  MoveL 6540 to (-70.92, -30.3, -10) mm, rotated rx 180 ry 0 rz 90 deg; joints [72.111, -18.401, 88.578, 0, 19.823, 72.111]
  MoveC 6541 to (-72.65, -31.38, -10) mm, rotated rx 180 ry 0 rz 90 deg; joints [72.056, -18.422, 88.671, 0, 19.752, 72.056] to (-73.33, -33.3, -10) mm, rotated rx 180 ry 0 rz 90 deg; joints [71.985, -18.423, 88.674, 0, 19.749, 71.985]
  MoveL 6542 to (-73.33, -68.7, -10) mm, rotated rx 180 ry 0 rz 90 deg; joints [70.818, -18.238, 87.875, 0, 20.362, 70.818]
  MoveL 6543 to (-73.33, -69.73, -10) mm, rotated rx 180 ry 0 rz 90 deg; joints [70.785, -18.232, 87.851, 0, 20.381, 70.785]
  MoveC 6544 to (-72.43, -71.9, -10) mm, rotated rx -180 ry 0 rz 90 deg; joints [70.724, -18.206, 87.74, 0, 20.466, 70.724] to (-70.27, -72.81, -10) mm, rotated rx 180 ry 0 rz 90 deg; joints [70.719, -18.167, 87.574, 0, 20.593, 70.719]
  MoveL 6545 to (-69.65, -72.82, -10) mm, rotated rx 180 ry 0 rz 90 deg; joints [70.726, -18.157, 87.532, 0, 20.625, 70.726]
  MoveL 6546 to (-55.44, -72.67, -10) mm, rotated rx -180 ry 0 rz 90 deg; joints [70.891, -17.926, 86.573, 0, 21.353, 70.891]
  MoveL 6547 to (-54.49, -72.66, -10) mm, rotated rx -180 ry 0 rz 90 deg; joints [70.902, -17.91, 86.509, 0, 21.401, 70.902]
  MoveL 6548 to (-37.43, -72.45, -10) mm, rotated rx -180 ry 0 rz 90 deg; joints [71.098, -17.621, 85.344, 0, 22.277, 71.098]
  MoveL 6549 to (-36.13, -72.43, -10) mm, rotated rx 180 ry 0 rz 90 deg; joints [71.114, -17.599, 85.254, 0, 22.344, 71.114]
  MoveC 6550 to (-35.1, -72.24, -10) mm, rotated rx -180 ry 0 rz 90 deg; joints [71.131, -17.582, 85.188, 0, 22.394, 71.131] to (-34.2, -71.71, -10) mm, rotated rx -180 ry 0 rz 90 deg; joints [71.158, -17.569, 85.138, 0, 22.431, 71.158]
  MoveC 6551 to (-33.55, -70.97, -10) mm, rotated rx -180 ry 0 rz 90 deg; joints [71.188, -17.562, 85.111, 0, 22.452, 71.188] to (-33.16, -70.08, -10) mm, rotated rx 180 ry 0 rz 90 deg; joints [71.221, -17.561, 85.105, 0, 22.456, 71.221]
  MoveL 6552 to (-21.39, -24.64, -10) mm, rotated rx 180 ry 0 rz 90 deg; joints [72.81, -17.613, 85.312, 0, 22.301, 72.81]
  MoveL 6553 to (-21.34, -24.17, -10) mm, rotated rx 180 ry 0 rz 90 deg; joints [72.826, -17.615, 85.319, 0, 22.296, 72.826]
  MoveC 6554 to (-22.27, -22.08, -10) mm, rotated rx -180 ry 0 rz 90 deg; joints [72.884, -17.642, 85.428, 0, 22.214, 72.884] to (-24.17, -20.81, -10) mm, rotated rx 180 ry 0 rz 90 deg; joints [72.906, -17.682, 85.587, 0, 22.095, 72.906]
  MoveC 6555 to (-24.63, -20.72, -10) mm, rotated rx -180 ry 0 rz 90 deg; joints [72.905, -17.691, 85.622, 0, 22.069, 72.905] to (-25.11, -20.75, -10) mm, rotated rx 180 ry 0 rz 90 deg; joints [72.899, -17.699, 85.655, 0, 22.045, 72.899]
  MoveL 6556 to (-31.75, -22.12, -10) mm, rotated rx 180 ry 0 rz 90 deg; joints [72.788, -17.806, 86.085, 0, 21.721, 72.788]
  MoveL 6557 to (-48.02, -25.51, -10) mm, rotated rx 180 ry 0 rz 90 deg; joints [72.51, -18.061, 87.131, 0, 20.93, 72.51]
  MoveL 6558 to (-46.48, -32.9, -10) mm, rotated rx 180 ry 0 rz 90 deg; joints [72.284, -17.997, 86.865, 0, 21.132, 72.284]
  MoveL 6559 to (-46.48, -32.9, -7) mm, rotated rx 180 ry 0 rz 90 deg; joints [72.284, -18.152, 86.967, 0, 21.185, 72.284]
  Establecer velocidad (1000.0 mm/s)
  MoveL 6560 to (-46.48, -32.9, 10) mm, rotated rx 180 ry 0 rz 90 deg; joints [72.284, -19.031, 87.535, 0, 21.495, 72.284]
  Establecer velocidad (66.7 mm/s)
  MoveL 6561 to (15.27, -63.53, 10) mm, rotated rx 180 ry 0 rz 90 deg; joints [71.941, -17.71, 82.508, 0, 25.202, 71.941]
  MoveL 6562 to (15.27, -63.53, -6.75) mm, rotated rx 180 ry 0 rz 90 deg; joints [71.941, -16.862, 81.946, 0, 24.916, 71.941]
  MoveL 6563 to (15.14, -65.04, -7.16) mm, rotated rx -180 ry 0 rz 90 deg; joints [71.892, -16.834, 81.906, 0, 24.928, 71.892]
  MoveL 6564 to (15.37, -66.54, -7.56) mm, rotated rx -180 ry 0 rz 90 deg; joints [71.847, -16.8, 81.84, 0, 24.959, 71.847]
  MoveL 6565 to (15.92, -67.95, -7.97) mm, rotated rx -180 ry 0 rz 90 deg; joints [71.809, -16.759, 81.753, 0, 25.006, 71.809]
  MoveL 6566 to (16.78, -69.21, -8.37) mm, rotated rx 180 ry 0 rz 90 deg; joints [71.778, -16.713, 81.647, 0, 25.066, 71.778]
  MoveL 6567 to (17.89, -70.24, -8.78) mm, rotated rx 180 ry 0 rz 90 deg; joints [71.758, -16.663, 81.528, 0, 25.135, 71.758]
  MoveL 6568 to (19.21, -71.01, -9.19) mm, rotated rx -180 ry 0 rz 90 deg; joints [71.747, -16.611, 81.401, 0, 25.21, 71.747]
  MoveL 6569 to (20.66, -71.46, -9.59) mm, rotated rx 180 ry 0 rz 90 deg; joints [71.748, -16.559, 81.271, 0, 25.287, 71.748]
  MoveL 6570 to (22.17, -71.55, -10) mm, rotated rx 180 ry 0 rz 90 deg; joints [71.761, -16.507, 81.145, 0, 25.362, 71.761]
  MoveC 6571 to (32.54, -71.19, -10) mm, rotated rx -180 ry 0 rz 90 deg; joints [71.878, -16.297, 80.397, 0, 25.9, 71.878] to (42.91, -70.78, -10) mm, rotated rx -180 ry 0 rz 90 deg; joints [71.995, -16.083, 79.643, 0, 26.44, 71.995]
  MoveC 6572 to (45.2, -67.86, -10) mm, rotated rx -180 ry 0 rz 90 deg; joints [72.108, -16.055, 79.544, 0, 26.51, 72.108] to (45.35, -64.16, -10) mm, rotated rx 180 ry 0 rz 90 deg; joints [72.224, -16.077, 79.621, 0, 26.455, 72.224]
  MoveC 6573 to (34.71, -51.22, -10) mm, rotated rx -180 ry 0 rz 90 deg; joints [72.521, -16.385, 80.708, 0, 25.677, 72.521] to (23.95, -38.38, -10) mm, rotated rx -180 ry 0 rz 90 deg; joints [72.819, -16.684, 81.785, 0, 24.899, 72.819]
  MoveL 6574 to (22.88, -37.43, -10) mm, rotated rx 180 ry 0 rz 90 deg; joints [72.838, -16.711, 81.884, 0, 24.827, 72.838]
  MoveL 6575 to (21.72, -36.48, -10) mm, rotated rx 180 ry 0 rz 90 deg; joints [72.857, -16.739, 81.989, 0, 24.75, 72.857]
  MoveL 6576 to (13.74, -29.98, -10) mm, rotated rx -180 ry 0 rz 90 deg; joints [72.986, -16.934, 82.708, 0, 24.226, 72.986]
  MoveL 6577 to (13.21, -29.55, -10) mm, rotated rx 180 ry 0 rz 90 deg; joints [72.994, -16.947, 82.756, 0, 24.191, 72.994]
  MoveC 6578 to (10.33, -29.1, -10) mm, rotated rx 180 ry 0 rz 90 deg; joints [72.98, -17.005, 82.972, 0, 24.033, 72.98] to (7.97, -30.8, -10) mm, rotated rx 180 ry 0 rz 90 deg; joints [72.903, -17.04, 83.104, 0, 23.936, 72.903]
  MoveL 6579 to (7.68, -31.75, -10) mm, rotated rx 180 ry 0 rz 90 deg; joints [72.87, -17.04, 83.104, 0, 23.936, 72.87]
  MoveL 6580 to (-2.03, -67.76, -10) mm, rotated rx -180 ry 0 rz 90 deg; joints [71.628, -17.006, 82.975, 0, 24.031, 71.628]
  MoveL 6581 to (-2.14, -68.23, -10) mm, rotated rx 180 ry 0 rz 90 deg; joints [71.612, -17.005, 82.971, 0, 24.034, 71.612]
  MoveC 6582 to (-1.24, -70.97, -10) mm, rotated rx 180 ry 0 rz 90 deg; joints [71.535, -16.97, 82.842, 0, 24.128, 71.535] to (1.42, -72.1, -10) mm, rotated rx 180 ry 0 rz 90 deg; joints [71.528, -16.912, 82.626, 0, 24.286, 71.528]
  MoveC 6583 to (11.8, -71.85, -10) mm, rotated rx 180 ry 0 rz 90 deg; joints [71.644, -16.712, 81.888, 0, 24.824, 71.644] to (22.17, -71.55, -10) mm, rotated rx 180 ry 0 rz 90 deg; joints [71.761, -16.507, 81.145, 0, 25.362, 71.761]
  MoveL 6584 to (21.93, -64.01, -10) mm, rotated rx 180 ry 0 rz 90 deg; joints [71.994, -16.561, 81.342, 0, 25.22, 71.994]
  MoveL 6585 to (21.93, -64.01, -7) mm, rotated rx -180 ry 0 rz 90 deg; joints [71.994, -16.713, 81.444, 0, 25.269, 71.994]
  Establecer velocidad (1000.0 mm/s)
  MoveL 6586 to (21.93, -64.01, 10) mm, rotated rx 180 ry 0 rz 90 deg; joints [71.994, -17.572, 82.015, 0, 25.557, 71.994]
  Establecer velocidad (66.7 mm/s)
  MoveL 6587 to (35, 18.65, 10) mm, rotated rx 180 ry 0 rz 90 deg; joints [74.731, -17.808, 82.861, 0, 24.947, 74.731]
  MoveL 6588 to (35, 18.65, -6.75) mm, rotated rx 180 ry 0 rz 90 deg; joints [74.731, -16.959, 82.299, 0, 24.66, 74.731]
  MoveL 6589 to (35.18, 20.15, -7.16) mm, rotated rx -180 ry 0 rz 90 deg; joints [74.781, -16.943, 82.302, 0, 24.641, 74.781]
  MoveL 6590 to (34.99, 21.66, -7.56) mm, rotated rx -180 ry 0 rz 90 deg; joints [74.827, -16.934, 82.332, 0, 24.602, 74.827]
  MoveL 6591 to (34.47, 23.09, -7.97) mm, rotated rx -180 ry 0 rz 90 deg; joints [74.869, -16.931, 82.384, 0, 24.547, 74.869]
  MoveL 6592 to (33.65, 24.37, -8.37) mm, rotated rx 180 ry 0 rz 90 deg; joints [74.902, -16.934, 82.455, 0, 24.479, 74.902]
  MoveL 6593 to (32.57, 25.43, -8.78) mm, rotated rx 180 ry 0 rz 90 deg; joints [74.927, -16.94, 82.541, 0, 24.399, 74.927]
  MoveL 6594 to (31.28, 26.23, -9.19) mm, rotated rx -180 ry 0 rz 90 deg; joints [74.941, -16.949, 82.637, 0, 24.312, 74.941]
  MoveL 6595 to (29.84, 26.72, -9.59) mm, rotated rx -180 ry 0 rz 90 deg; joints [74.945, -16.959, 82.737, 0, 24.222, 74.945]
  MoveL 6596 to (28.33, 26.86, -10) mm, rotated rx -180 ry 0 rz 90 deg; joints [74.936, -16.968, 82.835, 0, 24.133, 74.936]
  MoveC 6597 to (20.56, 26.8, -10) mm, rotated rx -180 ry 0 rz 90 deg; joints [74.867, -17.117, 83.395, 0, 23.723, 74.867] to (12.79, 26.71, -10) mm, rotated rx 180 ry 0 rz 90 deg; joints [74.796, -17.264, 83.95, 0, 23.313, 74.796]
  MoveC 6598 to (10.39, 25.38, -10) mm, rotated rx 180 ry 0 rz 90 deg; joints [74.731, -17.302, 84.096, 0, 23.205, 74.731] to (9.6, 22.74, -10) mm, rotated rx 180 ry 0 rz 90 deg; joints [74.639, -17.303, 84.101, 0, 23.202, 74.639]
  MoveL 6599 to (9.74, 22.27, -10) mm, rotated rx 180 ry 0 rz 90 deg; joints [74.625, -17.298, 84.082, 0, 23.216, 74.625]
  MoveL 6600 to (13.74, 11.38, -10) mm, rotated rx -180 ry 0 rz 90 deg; joints [74.309, -17.166, 83.579, 0, 23.587, 74.309]
  MoveL 6601 to (13.93, 10.89, -10) mm, rotated rx 180 ry 0 rz 90 deg; joints [74.295, -17.16, 83.556, 0, 23.604, 74.295]
  MoveC 6602 to (14.41, 10.01, -10) mm, rotated rx 180 ry 0 rz 90 deg; joints [74.271, -17.146, 83.504, 0, 23.643, 74.271] to (15.12, 9.3, -10) mm, rotated rx 180 ry 0 rz 90 deg; joints [74.255, -17.129, 83.438, 0, 23.691, 74.255]
  MoveL 6603 to (27.96, -0.34, -10) mm, rotated rx 180 ry 0 rz 90 deg; joints [74.063, -16.828, 82.315, 0, 24.513, 74.063]
  MoveL 6604 to (28.42, -0.67, -10) mm, rotated rx 180 ry 0 rz 90 deg; joints [74.056, -16.817, 82.274, 0, 24.543, 74.056]
  MoveC 6605 to (29.07, -1.02, -10) mm, rotated rx 180 ry 0 rz 90 deg; joints [74.051, -16.802, 82.22, 0, 24.583, 74.051] to (29.8, -1.18, -10) mm, rotated rx 180 ry 0 rz 90 deg; joints [74.053, -16.787, 82.164, 0, 24.623, 74.053]
  MoveC 6606 to (31.81, -0.82, -10) mm, rotated rx -180 ry 0 rz 90 deg; joints [74.082, -16.749, 82.025, 0, 24.724, 74.082] to (33.4, 0.47, -10) mm, rotated rx 180 ry 0 rz 90 deg; joints [74.138, -16.725, 81.936, 0, 24.789, 74.138]
  MoveL 6607 to (45.89, 18.48, -10) mm, rotated rx -180 ry 0 rz 90 deg; joints [74.82, -16.574, 81.388, 0, 25.187, 74.82]
  MoveL 6608 to (47.25, 20.51, -10) mm, rotated rx 180 ry 0 rz 90 deg; joints [74.896, -16.557, 81.327, 0, 25.23, 74.896]
  MoveC 6609 to (47.11, 23.56, -10) mm, rotated rx 180 ry 0 rz 90 deg; joints [74.992, -16.577, 81.398, 0, 25.179, 74.992] to (45.53, 26.17, -10) mm, rotated rx 180 ry 0 rz 90 deg; joints [75.062, -16.623, 81.566, 0, 25.057, 75.062]
  MoveC 6610 to (44.76, 26.68, -10) mm, rotated rx 180 ry 0 rz 90 deg; joints [75.071, -16.642, 81.633, 0, 25.009, 75.071] to (43.86, 26.86, -10) mm, rotated rx -180 ry 0 rz 90 deg; joints [75.069, -16.661, 81.702, 0, 24.959, 75.069]
  MoveC 6611 to (36.09, 26.87, -10) mm, rotated rx 180 ry 0 rz 90 deg; joints [75.004, -16.816, 82.271, 0, 24.545, 75.004] to (28.33, 26.86, -10) mm, rotated rx -180 ry 0 rz 90 deg; joints [74.936, -16.968, 82.835, 0, 24.133, 74.936]
  MoveL 6612 to (28.36, 19.31, -10) mm, rotated rx 180 ry 0 rz 90 deg; joints [74.694, -16.928, 82.684, 0, 24.244, 74.694]
  MoveL 6613 to (28.36, 19.31, -7) mm, rotated rx 180 ry 0 rz 90 deg; joints [74.694, -17.08, 82.786, 0, 24.294, 74.694]
  Establecer velocidad (1000.0 mm/s)
  MoveL 6614 to (28.36, 19.31, 10) mm, rotated rx 180 ry 0 rz 90 deg; joints [74.694, -17.944, 83.356, 0, 24.588, 74.694]
  Establecer velocidad (66.7 mm/s)
  MoveL 6615 to (6.83, 65.57, 10) mm, rotated rx 180 ry 0 rz 90 deg; joints [76.013, -18.584, 85.767, 0, 22.817, 76.013]
  MoveL 6616 to (6.83, 65.57, -6.75) mm, rotated rx -180 ry 0 rz 90 deg; joints [76.013, -17.726, 85.207, 0, 22.518, 76.013]
  MoveL 6617 to (6.78, 64.06, -7.16) mm, rotated rx 180 ry 0 rz 90 deg; joints [75.963, -17.699, 85.17, 0, 22.529, 75.963]
  MoveL 6618 to (7.11, 62.57, -7.56) mm, rotated rx 180 ry 0 rz 90 deg; joints [75.917, -17.665, 85.107, 0, 22.559, 75.917]
  MoveL 6619 to (7.75, 61.2, -7.97) mm, rotated rx -180 ry 0 rz 90 deg; joints [75.877, -17.626, 85.022, 0, 22.604, 75.877]
  MoveL 6620 to (8.69, 59.99, -8.37) mm, rotated rx -180 ry 0 rz 90 deg; joints [75.845, -17.583, 84.921, 0, 22.662, 75.845]
  MoveL 6621 to (9.86, 59.03, -8.78) mm, rotated rx 180 ry 0 rz 90 deg; joints [75.824, -17.537, 84.806, 0, 22.731, 75.824]
  MoveL 6622 to (11.22, 58.35, -9.19) mm, rotated rx 180 ry 0 rz 90 deg; joints [75.813, -17.488, 84.683, 0, 22.805, 75.813]
  MoveL 6623 to (12.7, 57.99, -9.59) mm, rotated rx -180 ry 0 rz 90 deg; joints [75.813, -17.438, 84.557, 0, 22.881, 75.813]
  MoveL 6624 to (14.21, 58, -10) mm, rotated rx 180 ry 0 rz 90 deg; joints [75.826, -17.389, 84.435, 0, 22.954, 75.826]
  MoveL 6625 to (16.31, 58.19, -10) mm, rotated rx 180 ry 0 rz 90 deg; joints [75.849, -17.352, 84.289, 0, 23.063, 75.849]
  MoveC 6626 to (25.93, 59.17, -10) mm, rotated rx -180 ry 0 rz 90 deg; joints [75.96, -17.176, 83.615, 0, 23.561, 75.96] to (35.54, 60.24, -10) mm, rotated rx -180 ry 0 rz 90 deg; joints [76.072, -16.996, 82.938, 0, 24.058, 76.072]
  MoveC 6627 to (46.2, 61.66, -10) mm, rotated rx -180 ry 0 rz 90 deg; joints [76.202, -16.793, 82.185, 0, 24.608, 76.202] to (56.82, 63.37, -10) mm, rotated rx 180 ry 0 rz 90 deg; joints [76.34, -16.586, 81.432, 0, 25.154, 76.34]
  MoveL 6628 to (56.82, 69.31, -10) mm, rotated rx 180 ry 0 rz 90 deg; joints [76.531, -16.616, 81.538, 0, 25.077, 76.531]
  MoveC 6629 to (39.09, 70.56, -10) mm, rotated rx 180 ry 0 rz 90 deg; joints [76.434, -16.976, 82.864, 0, 24.112, 76.434] to (21.32, 71.33, -10) mm, rotated rx -180 ry 0 rz 90 deg; joints [76.319, -17.319, 84.163, 0, 23.156, 76.319]
  MoveC 6630 to (0.83, 71.9, -10) mm, rotated rx -180 ry 0 rz 90 deg; joints [76.173, -17.694, 85.632, 0, 22.061, 76.173] to (-19.66, 72.35, -10) mm, rotated rx 180 ry 0 rz 90 deg; joints [76.019, -18.048, 87.076, 0, 20.972, 76.019]
  MoveC 6631 to (-22, 69.47, -10) mm, rotated rx -180 ry 0 rz 90 deg; joints [75.904, -18.075, 87.189, 0, 20.886, 75.904] to (-21.68, 65.78, -10) mm, rotated rx 180 ry 0 rz 90 deg; joints [75.783, -18.054, 87.103, 0, 20.952, 75.783]
  MoveL 6632 to (-7.47, 56.63, -10) mm, rotated rx 180 ry 0 rz 90 deg; joints [75.599, -17.772, 85.947, 0, 21.825, 75.599]
  MoveC 6633 to (-7.12, 56.43, -10) mm, rotated rx 180 ry 0 rz 90 deg; joints [75.596, -17.765, 85.919, 0, 21.846, 75.596] to (-6.75, 56.27, -10) mm, rotated rx -180 ry 0 rz 90 deg; joints [75.594, -17.758, 85.89, 0, 21.868, 75.594]
  MoveC 6634 to (4.78, 57.16, -10) mm, rotated rx 180 ry 0 rz 90 deg; joints [75.72, -17.557, 85.092, 0, 22.466, 75.72] to (16.31, 58.19, -10) mm, rotated rx 180 ry 0 rz 90 deg; joints [75.849, -17.352, 84.289, 0, 23.063, 75.849]
  MoveL 6635 to (15.59, 65.71, -10) mm, rotated rx 180 ry 0 rz 90 deg; joints [76.089, -17.4, 84.475, 0, 22.925, 76.089]
  MoveL 6636 to (0.19, 64.36, -10) mm, rotated rx 180 ry 0 rz 90 deg; joints [75.919, -17.672, 85.546, 0, 22.126, 75.919]
  MoveL 6637 to (0.19, 64.36, -7) mm, rotated rx 180 ry 0 rz 90 deg; joints [75.919, -17.826, 85.648, 0, 22.179, 75.919]
  Establecer velocidad (1000.0 mm/s)
  MoveL 6638 to (0.19, 64.36, 10) mm, rotated rx -180 ry 0 rz 90 deg; joints [75.919, -18.7, 86.216, 0, 22.484, 75.919]
  Establecer velocidad (66.7 mm/s)
  MoveL 6639 to (3.74, 65.44, 10) mm, rotated rx -180 ry 0 rz 90 deg; joints [75.983, -18.64, 85.984, 0, 22.656, 75.983]
  MoveL 6640 to (3.74, 65.44, -7) mm, rotated rx -180 ry 0 rz 90 deg; joints [75.983, -17.768, 85.415, 0, 22.352, 75.983]
  MoveL 6641 to (3.7, 63.92, -7.41) mm, rotated rx -180 ry 0 rz 90 deg; joints [75.933, -17.741, 85.378, 0, 22.363, 75.933]
  MoveL 6642 to (4.03, 62.44, -7.81) mm, rotated rx 180 ry 0 rz 90 deg; joints [75.887, -17.707, 85.314, 0, 22.393, 75.887]
  MoveL 6643 to (4.67, 61.06, -8.22) mm, rotated rx -180 ry 0 rz 90 deg; joints [75.847, -17.669, 85.23, 0, 22.438, 75.847]
  MoveL 6644 to (5.61, 59.86, -8.63) mm, rotated rx 180 ry 0 rz 90 deg; joints [75.816, -17.625, 85.129, 0, 22.497, 75.816]
  MoveL 6645 to (6.78, 58.9, -9.03) mm, rotated rx -180 ry 0 rz 90 deg; joints [75.794, -17.579, 85.014, 0, 22.565, 75.794]
  MoveL 6646 to (8.14, 58.22, -9.44) mm, rotated rx 180 ry 0 rz 90 deg; joints [75.783, -17.53, 84.891, 0, 22.639, 75.783]
  MoveL 6647 to (9.62, 57.86, -9.84) mm, rotated rx 180 ry 0 rz 90 deg; joints [75.783, -17.481, 84.766, 0, 22.715, 75.783]
  MoveL 6648 to (11.13, 57.87, -10.25) mm, rotated rx -180 ry 0 rz 90 deg; joints [75.796, -17.433, 84.644, 0, 22.788, 75.796]
  MoveL 6649 to (16.29, 58.36, -10.25) mm, rotated rx -180 ry 0 rz 90 deg; joints [75.855, -17.34, 84.285, 0, 23.055, 75.855]
  MoveC 6650 to (25.45, 59.31, -10.25) mm, rotated rx -180 ry 0 rz 90 deg; joints [75.96, -17.173, 83.644, 0, 23.529, 75.96] to (34.59, 60.34, -10.25) mm, rotated rx -180 ry 0 rz 90 deg; joints [76.068, -17.002, 83, 0, 24.002, 76.068]
  MoveC 6651 to (44.29, 61.63, -10.25) mm, rotated rx -180 ry 0 rz 90 deg; joints [76.187, -16.818, 82.315, 0, 24.502, 76.187] to (53.96, 63.16, -10.25) mm, rotated rx -180 ry 0 rz 90 deg; joints [76.312, -16.631, 81.631, 0, 25, 76.312]
  MoveL 6652 to (53.96, 69.23, -10.25) mm, rotated rx 180 ry 0 rz 90 deg; joints [76.506, -16.661, 81.74, 0, 24.921, 76.506]
  MoveC 6653 to (38.5, 70.34, -10.25) mm, rotated rx -180 ry 0 rz 90 deg; joints [76.422, -16.974, 82.894, 0, 24.08, 76.422] to (23.02, 71.05, -10.25) mm, rotated rx -180 ry 0 rz 90 deg; joints [76.323, -17.273, 84.027, 0, 23.246, 76.323]
  MoveC 6654 to (1.99, 71.66, -10.25) mm, rotated rx -180 ry 0 rz 90 deg; joints [76.174, -17.659, 85.538, 0, 22.121, 76.174] to (-19.04, 72.14, -10.25) mm, rotated rx 180 ry 0 rz 90 deg; joints [76.017, -18.024, 87.021, 0, 21.002, 76.017]
  MoveC 6655 to (-21.35, 69.3, -10.25) mm, rotated rx -180 ry 0 rz 90 deg; joints [75.903, -18.051, 87.132, 0, 20.918, 75.903] to (-21.05, 65.65, -10.25) mm, rotated rx 180 ry 0 rz 90 deg; joints [75.784, -18.03, 87.048, 0, 20.983, 75.784]
  MoveL 6656 to (-6.9, 56.54, -10.25) mm, rotated rx 180 ry 0 rz 90 deg; joints [75.601, -17.749, 85.897, 0, 21.852, 75.601]
  MoveC 6657 to (-6.66, 56.43, -10.25) mm, rotated rx 180 ry 0 rz 90 deg; joints [75.6, -17.744, 85.878, 0, 21.866, 75.6] to (-6.41, 56.41, -10.25) mm, rotated rx 180 ry 0 rz 90 deg; joints [75.601, -17.74, 85.86, 0, 21.88, 75.601]
  MoveC 6658 to (4.95, 57.32, -10.25) mm, rotated rx -180 ry 0 rz 90 deg; joints [75.726, -17.542, 85.074, 0, 22.468, 75.726] to (16.29, 58.36, -10.25) mm, rotated rx -180 ry 0 rz 90 deg; joints [75.855, -17.34, 84.285, 0, 23.055, 75.855]
  MoveL 6659 to (15.55, 65.87, -10.25) mm, rotated rx 180 ry 0 rz 90 deg; joints [76.094, -17.388, 84.472, 0, 22.916, 76.094]
  MoveL 6660 to (-3.03, 64.24, -10.25) mm, rotated rx 180 ry 0 rz 90 deg; joints [75.888, -17.715, 85.762, 0, 21.953, 75.888]
  MoveL 6661 to (-3.03, 64.24, -7.25) mm, rotated rx 180 ry 0 rz 90 deg; joints [75.888, -17.87, 85.864, 0, 22.006, 75.888]
  Establecer velocidad (1000.0 mm/s)
  MoveL 6662 to (-3.03, 64.24, 10) mm, rotated rx -180 ry 0 rz 90 deg; joints [75.888, -18.757, 86.441, 0, 22.316, 75.888]
  Establecer velocidad (66.7 mm/s)
  MoveL 6663 to (35.09, 18.39, 10) mm, rotated rx 180 ry 0 rz 90 deg; joints [74.724, -17.805, 82.849, 0, 24.956, 74.724]
  MoveL 6664 to (35.09, 18.39, -7) mm, rotated rx -180 ry 0 rz 90 deg; joints [74.724, -16.943, 82.279, 0, 24.664, 74.724]
  MoveL 6665 to (35.27, 19.9, -7.41) mm, rotated rx -180 ry 0 rz 90 deg; joints [74.773, -16.927, 82.282, 0, 24.645, 74.773]
  MoveL 6666 to (35.09, 21.41, -7.81) mm, rotated rx 180 ry 0 rz 90 deg; joints [74.82, -16.918, 82.312, 0, 24.607, 74.82]
  MoveL 6667 to (34.57, 22.84, -8.22) mm, rotated rx -180 ry 0 rz 90 deg; joints [74.861, -16.915, 82.363, 0, 24.552, 74.861]
  MoveL 6668 to (33.75, 24.12, -8.63) mm, rotated rx -180 ry 0 rz 90 deg; joints [74.895, -16.918, 82.435, 0, 24.483, 74.895]
  MoveL 6669 to (32.67, 25.19, -9.03) mm, rotated rx -180 ry 0 rz 90 deg; joints [74.92, -16.924, 82.52, 0, 24.404, 74.92]
  MoveL 6670 to (31.38, 25.99, -9.44) mm, rotated rx 180 ry 0 rz 90 deg; joints [74.935, -16.933, 82.616, 0, 24.317, 74.935]
  MoveL 6671 to (29.94, 26.48, -9.84) mm, rotated rx 180 ry 0 rz 90 deg; joints [74.938, -16.943, 82.716, 0, 24.227, 74.938]
  MoveL 6672 to (28.43, 26.62, -10.25) mm, rotated rx -180 ry 0 rz 90 deg; joints [74.929, -16.952, 82.815, 0, 24.138, 74.929]
  MoveC 6673 to (21.08, 26.58, -10.25) mm, rotated rx -180 ry 0 rz 90 deg; joints [74.864, -17.094, 83.344, 0, 23.749, 74.864] to (13.74, 26.52, -10.25) mm, rotated rx 180 ry 0 rz 90 deg; joints [74.798, -17.232, 83.87, 0, 23.362, 74.798]
  MoveL 6674 to (12.79, 26.47, -10.25) mm, rotated rx 180 ry 0 rz 90 deg; joints [74.788, -17.25, 83.937, 0, 23.312, 74.788]
  MoveC 6675 to (10.55, 25.01, -10.25) mm, rotated rx 180 ry 0 rz 90 deg; joints [74.721, -17.284, 84.069, 0, 23.215, 74.721] to (9.95, 22.4, -10.25) mm, rotated rx -180 ry 0 rz 90 deg; joints [74.631, -17.282, 84.061, 0, 23.221, 74.631]
  MoveL 6676 to (9.99, 22.27, -10.25) mm, rotated rx 180 ry 0 rz 90 deg; joints [74.627, -17.28, 84.055, 0, 23.225, 74.627]
  MoveL 6677 to (13.82, 11.85, -10.25) mm, rotated rx -180 ry 0 rz 90 deg; joints [74.325, -17.154, 83.574, 0, 23.58, 74.325]
  MoveL 6678 to (14.18, 10.92, -10.25) mm, rotated rx 180 ry 0 rz 90 deg; joints [74.298, -17.143, 83.53, 0, 23.612, 74.298]
  MoveC 6679 to (14.61, 10.13, -10.25) mm, rotated rx -180 ry 0 rz 90 deg; joints [74.277, -17.13, 83.483, 0, 23.647, 74.277] to (15.25, 9.5, -10.25) mm, rotated rx 180 ry 0 rz 90 deg; joints [74.262, -17.115, 83.425, 0, 23.69, 74.262]
  MoveL 6680 to (28.34, -0.31, -10.25) mm, rotated rx 180 ry 0 rz 90 deg; joints [74.067, -16.808, 82.279, 0, 24.529, 74.067]
  MoveC 6681 to (29.16, -0.73, -10.25) mm, rotated rx -180 ry 0 rz 90 deg; joints [74.061, -16.789, 82.211, 0, 24.579, 74.061] to (30.08, -0.84, -10.25) mm, rotated rx 180 ry 0 rz 90 deg; joints [74.066, -16.771, 82.142, 0, 24.629, 74.066]
  MoveL 6682 to (30.41, -0.82, -10.25) mm, rotated rx 180 ry 0 rz 90 deg; joints [74.07, -16.764, 82.118, 0, 24.646, 74.07]
  MoveC 6683 to (32.1, -0.33, -10.25) mm, rotated rx 180 ry 0 rz 90 deg; joints [74.101, -16.734, 82.006, 0, 24.728, 74.101] to (33.39, 0.86, -10.25) mm, rotated rx 180 ry 0 rz 90 deg; joints [74.15, -16.715, 81.936, 0, 24.779, 74.15]
  MoveL 6684 to (45.56, 18.48, -10.25) mm, rotated rx -180 ry 0 rz 90 deg; joints [74.817, -16.568, 81.403, 0, 25.165, 74.817]
  MoveL 6685 to (46.21, 19.43, -10.25) mm, rotated rx -180 ry 0 rz 90 deg; joints [74.853, -16.56, 81.374, 0, 25.186, 74.853]
  MoveL 6686 to (46.79, 20.37, -10.25) mm, rotated rx -180 ry 0 rz 90 deg; joints [74.888, -16.553, 81.35, 0, 25.203, 74.888]
  MoveC 6687 to (46.42, 23.91, -10.25) mm, rotated rx -180 ry 0 rz 90 deg; joints [74.997, -16.58, 81.448, 0, 25.133, 74.997] to (44.07, 26.58, -10.25) mm, rotated rx 180 ry 0 rz 90 deg; joints [75.062, -16.643, 81.673, 0, 24.97, 75.062]
  MoveC 6688 to (36.25, 26.62, -10.25) mm, rotated rx -180 ry 0 rz 90 deg; joints [74.997, -16.799, 82.246, 0, 24.553, 74.997] to (28.43, 26.62, -10.25) mm, rotated rx -180 ry 0 rz 90 deg; joints [74.929, -16.952, 82.815, 0, 24.138, 74.929]
  MoveL 6689 to (28.45, 19.07, -10.25) mm, rotated rx -180 ry 0 rz 90 deg; joints [74.687, -16.912, 82.664, 0, 24.248, 74.687]
  MoveL 6690 to (28.45, 19.07, -7.25) mm, rotated rx -180 ry 0 rz 90 deg; joints [74.687, -17.065, 82.767, 0, 24.298, 74.687]
  Establecer velocidad (1000.0 mm/s)
  MoveL 6691 to (28.45, 19.07, 10) mm, rotated rx -180 ry 0 rz 90 deg; joints [74.687, -17.941, 83.345, 0, 24.596, 74.687]
  Establecer velocidad (66.7 mm/s)
  MoveL 6692 to (15.14, -63.32, 10) mm, rotated rx -180 ry 0 rz 90 deg; joints [71.946, -17.714, 82.522, 0, 25.192, 71.946]
  MoveL 6693 to (15.14, -63.32, -7) mm, rotated rx -180 ry 0 rz 90 deg; joints [71.946, -16.853, 81.952, 0, 24.902, 71.946]
  MoveL 6694 to (15, -64.83, -7.41) mm, rotated rx -180 ry 0 rz 90 deg; joints [71.897, -16.826, 81.912, 0, 24.914, 71.897]
  MoveL 6695 to (15.23, -66.33, -7.81) mm, rotated rx -180 ry 0 rz 90 deg; joints [71.853, -16.791, 81.846, 0, 24.945, 71.853]
  MoveL 6696 to (15.8, -67.74, -8.22) mm, rotated rx 180 ry 0 rz 90 deg; joints [71.814, -16.75, 81.758, 0, 24.991, 71.814]
  MoveL 6697 to (16.65, -69, -8.63) mm, rotated rx 180 ry 0 rz 90 deg; joints [71.784, -16.704, 81.653, 0, 25.051, 71.784]
  MoveL 6698 to (17.77, -70.03, -9.03) mm, rotated rx -180 ry 0 rz 90 deg; joints [71.763, -16.654, 81.534, 0, 25.121, 71.763]
  MoveL 6699 to (19.08, -70.79, -9.44) mm, rotated rx 180 ry 0 rz 90 deg; joints [71.753, -16.602, 81.406, 0, 25.196, 71.753]
  MoveL 6700 to (20.53, -71.24, -9.84) mm, rotated rx 180 ry 0 rz 90 deg; joints [71.754, -16.55, 81.277, 0, 25.273, 71.754]
  MoveL 6701 to (22.05, -71.33, -10.25) mm, rotated rx -180 ry 0 rz 90 deg; joints [71.766, -16.498, 81.151, 0, 25.347, 71.766]
  MoveC 6702 to (32.24, -70.96, -10.25) mm, rotated rx 180 ry 0 rz 90 deg; joints [71.882, -16.293, 80.416, 0, 25.876, 71.882] to (42.43, -70.52, -10.25) mm, rotated rx 180 ry 0 rz 90 deg; joints [71.998, -16.082, 79.677, 0, 26.406, 71.998]
  MoveC 6703 to (44.68, -67.63, -10.25) mm, rotated rx 180 ry 0 rz 90 deg; joints [72.11, -16.055, 79.579, 0, 26.475, 72.11] to (44.82, -63.97, -10.25) mm, rotated rx 180 ry 0 rz 90 deg; joints [72.225, -16.077, 79.657, 0, 26.42, 72.225]
  MoveL 6704 to (44.11, -63.02, -10.25) mm, rotated rx -180 ry 0 rz 90 deg; joints [72.247, -16.098, 79.732, 0, 26.366, 72.247]
  MoveL 6705 to (37.89, -55.44, -10.25) mm, rotated rx 180 ry 0 rz 90 deg; joints [72.421, -16.279, 80.368, 0, 25.911, 72.421]
  MoveL 6706 to (24.12, -38.91, -10.25) mm, rotated rx 180 ry 0 rz 90 deg; joints [72.804, -16.664, 81.752, 0, 24.912, 72.804]
  MoveC 6707 to (23.68, -38.42, -10.25) mm, rotated rx -180 ry 0 rz 90 deg; joints [72.815, -16.676, 81.795, 0, 24.881, 72.815] to (23.2, -37.98, -10.25) mm, rotated rx 180 ry 0 rz 90 deg; joints [72.824, -16.688, 81.84, 0, 24.848, 72.824]
  MoveL 6708 to (22.54, -37.43, -10.25) mm, rotated rx -180 ry 0 rz 90 deg; joints [72.835, -16.705, 81.9, 0, 24.805, 72.835]
  MoveL 6709 to (13.27, -29.86, -10.25) mm, rotated rx -180 ry 0 rz 90 deg; joints [72.985, -16.932, 82.737, 0, 24.195, 72.985]
  MoveC 6710 to (11.38, -29.38, -10.25) mm, rotated rx 180 ry 0 rz 90 deg; joints [72.981, -16.971, 82.882, 0, 24.088, 72.981] to (9.49, -29.85, -10.25) mm, rotated rx -180 ry 0 rz 90 deg; joints [72.948, -17.004, 83.008, 0, 23.997, 72.948]
  MoveL 6711 to (9.16, -30.03, -10.25) mm, rotated rx 180 ry 0 rz 90 deg; joints [72.939, -17.009, 83.028, 0, 23.982, 72.939]
  MoveC 6712 to (8.42, -30.65, -10.25) mm, rotated rx 180 ry 0 rz 90 deg; joints [72.912, -17.02, 83.067, 0, 23.953, 72.912] to (7.99, -31.51, -10.25) mm, rotated rx 180 ry 0 rz 90 deg; joints [72.88, -17.023, 83.079, 0, 23.944, 72.88]
  MoveL 6713 to (-1.55, -66.81, -10.25) mm, rotated rx -180 ry 0 rz 90 deg; joints [71.663, -16.99, 82.954, 0, 24.036, 71.663]
  MoveL 6714 to (-1.89, -68.23, -10.25) mm, rotated rx -180 ry 0 rz 90 deg; joints [71.615, -16.987, 82.945, 0, 24.043, 71.615]
  MoveC 6715 to (-0.91, -70.83, -10.25) mm, rotated rx 180 ry 0 rz 90 deg; joints [71.543, -16.952, 82.813, 0, 24.139, 71.543] to (1.66, -71.88, -10.25) mm, rotated rx 180 ry 0 rz 90 deg; joints [71.537, -16.896, 82.605, 0, 24.291, 71.537]
  MoveC 6716 to (11.86, -71.64, -10.25) mm, rotated rx -180 ry 0 rz 90 deg; joints [71.651, -16.699, 81.88, 0, 24.819, 71.651] to (22.05, -71.33, -10.25) mm, rotated rx -180 ry 0 rz 90 deg; joints [71.766, -16.498, 81.151, 0, 25.347, 71.766]
  MoveL 6717 to (21.8, -63.78, -10.25) mm, rotated rx -180 ry 0 rz 90 deg; joints [72, -16.553, 81.348, 0, 25.205, 72]
  MoveL 6718 to (21.8, -63.78, -7.25) mm, rotated rx -180 ry 0 rz 90 deg; joints [72, -16.705, 81.451, 0, 25.254, 72]
  Establecer velocidad (1000.0 mm/s)
  MoveL 6719 to (21.8, -63.78, 10) mm, rotated rx 180 ry 0 rz 90 deg; joints [72, -17.577, 82.03, 0, 25.546, 72]
  Establecer velocidad (66.7 mm/s)
  MoveL 6720 to (-37.16, -52.05, 10) mm, rotated rx -180 ry 0 rz 90 deg; joints [71.759, -18.764, 86.468, 0, 22.296, 71.759]
  MoveL 6721 to (-37.16, -52.05, -7) mm, rotated rx 180 ry 0 rz 90 deg; joints [71.759, -17.89, 85.9, 0, 21.99, 71.759]
  MoveL 6722 to (-35.75, -52.61, -7.41) mm, rotated rx -180 ry 0 rz 90 deg; joints [71.756, -17.841, 85.776, 0, 22.065, 71.756]
  MoveL 6723 to (-34.24, -52.81, -7.81) mm, rotated rx 180 ry 0 rz 90 deg; joints [71.766, -17.793, 85.654, 0, 22.139, 71.766]
  MoveL 6724 to (-32.73, -52.67, -8.22) mm, rotated rx 180 ry 0 rz 90 deg; joints [71.786, -17.746, 85.538, 0, 22.208, 71.786]
  MoveL 6725 to (-31.28, -52.2, -8.63) mm, rotated rx -180 ry 0 rz 90 deg; joints [71.817, -17.703, 85.435, 0, 22.268, 71.817]
  MoveL 6726 to (-29.97, -51.43, -9.03) mm, rotated rx -180 ry 0 rz 90 deg; joints [71.855, -17.664, 85.348, 0, 22.315, 71.855]
  MoveL 6727 to (-28.87, -50.38, -9.44) mm, rotated rx 180 ry 0 rz 90 deg; joints [71.901, -17.63, 85.282, 0, 22.348, 71.901]
  MoveL 6728 to (-28.03, -49.12, -9.84) mm, rotated rx -180 ry 0 rz 90 deg; joints [71.95, -17.601, 85.238, 0, 22.363, 71.95]
  MoveL 6729 to (-27.52, -47.69, -10.25) mm, rotated rx 180 ry 0 rz 90 deg; joints [72.002, -17.579, 85.221, 0, 22.359, 72.002]
  MoveL 6730 to (-21.66, -25.11, -10.25) mm, rotated rx 180 ry 0 rz 90 deg; joints [72.792, -17.603, 85.312, 0, 22.29, 72.792]
  MoveC 6731 to (-21.58, -24.64, -10.25) mm, rotated rx 180 ry 0 rz 90 deg; joints [72.808, -17.604, 85.316, 0, 22.287, 72.808] to (-21.6, -24.17, -10.25) mm, rotated rx 180 ry 0 rz 90 deg; joints [72.823, -17.606, 85.328, 0, 22.279, 72.823]
  MoveC 6732 to (-22.64, -22.11, -10.25) mm, rotated rx 180 ry 0 rz 90 deg; joints [72.88, -17.636, 85.445, 0, 22.191, 72.88] to (-24.64, -20.94, -10.25) mm, rotated rx -180 ry 0 rz 90 deg; joints [72.897, -17.677, 85.609, 0, 22.068, 72.897]
  MoveC 6733 to (-25.03, -20.94, -10.25) mm, rotated rx 180 ry 0 rz 90 deg; joints [72.894, -17.684, 85.636, 0, 22.048, 72.894] to (-25.41, -20.99, -10.25) mm, rotated rx -180 ry 0 rz 90 deg; joints [72.888, -17.69, 85.662, 0, 22.029, 72.888]
  MoveL 6734 to (-32.69, -22.48, -10.25) mm, rotated rx -180 ry 0 rz 90 deg; joints [72.766, -17.808, 86.135, 0, 21.673, 72.766]
  MoveL 6735 to (-70.75, -30.41, -10.25) mm, rotated rx 180 ry 0 rz 90 deg; joints [72.109, -18.385, 88.555, 0, 19.829, 72.109]
  MoveC 6736 to (-72.48, -31.47, -10.25) mm, rotated rx -180 ry 0 rz 90 deg; joints [72.055, -18.406, 88.649, 0, 19.757, 72.055] to (-73.16, -33.39, -10.25) mm, rotated rx 180 ry 0 rz 90 deg; joints [71.984, -18.407, 88.653, 0, 19.754, 71.984]
  MoveL 6737 to (-73.17, -68.7, -10.25) mm, rotated rx -180 ry 0 rz 90 deg; joints [70.82, -18.222, 87.856, 0, 20.366, 70.82]
  MoveL 6738 to (-73.16, -69.64, -10.25) mm, rotated rx 180 ry 0 rz 90 deg; joints [70.79, -18.217, 87.833, 0, 20.384, 70.79]
  MoveC 6739 to (-72.23, -71.81, -10.25) mm, rotated rx 180 ry 0 rz 90 deg; joints [70.729, -18.19, 87.721, 0, 20.47, 70.729] to (-70.05, -72.68, -10.25) mm, rotated rx 180 ry 0 rz 90 deg; joints [70.726, -18.151, 87.553, 0, 20.598, 70.726]
  MoveL 6740 to (-38.38, -72.3, -10.25) mm, rotated rx 180 ry 0 rz 90 deg; joints [71.093, -17.626, 85.404, 0, 22.221, 71.093]
  MoveL 6741 to (-36.21, -72.27, -10.25) mm, rotated rx 180 ry 0 rz 90 deg; joints [71.118, -17.588, 85.256, 0, 22.333, 71.118]
  MoveC 6742 to (-34.5, -71.7, -10.25) mm, rotated rx -180 ry 0 rz 90 deg; joints [71.155, -17.562, 85.15, 0, 22.411, 71.155] to (-33.41, -70.25, -10.25) mm, rotated rx 180 ry 0 rz 90 deg; joints [71.213, -17.551, 85.109, 0, 22.442, 71.213]
  MoveC 6743 to (-33.25, -69.79, -10.25) mm, rotated rx -180 ry 0 rz 90 deg; joints [71.23, -17.551, 85.109, 0, 22.442, 71.23] to (-33.12, -69.31, -10.25) mm, rotated rx 180 ry 0 rz 90 deg; joints [71.246, -17.552, 85.111, 0, 22.441, 71.246]
  MoveL 6744 to (-27.52, -47.69, -10.25) mm, rotated rx 180 ry 0 rz 90 deg; joints [72.002, -17.579, 85.221, 0, 22.359, 72.002]
  MoveL 6745 to (-34.82, -45.8, -10.25) mm, rotated rx -180 ry 0 rz 90 deg; joints [71.986, -17.717, 85.77, 0, 21.947, 71.986]
  MoveL 6746 to (-34.82, -45.8, -7.25) mm, rotated rx 180 ry 0 rz 90 deg; joints [71.986, -17.872, 85.872, 0, 22, 71.986]
  Establecer velocidad (1000.0 mm/s)
  MoveL 6747 to (-34.82, -45.8, 10) mm, rotated rx -180 ry 0 rz 90 deg; joints [71.986, -18.759, 86.449, 0, 22.31, 71.986]
  Establecer velocidad (66.7 mm/s)
  MoveL 6748 to (-64.93, 36.02, 10) mm, rotated rx 180 ry 0 rz 90 deg; joints [74.395, -19.659, 90.186, 0, 19.473, 74.395]
  MoveL 6749 to (-64.93, 36.02, -7) mm, rotated rx 180 ry 0 rz 90 deg; joints [74.395, -18.77, 89.618, 0, 19.152, 74.395]
  MoveL 6750 to (-66.43, 36.2, -7.41) mm, rotated rx 180 ry 0 rz 90 deg; joints [74.387, -18.772, 89.709, 0, 19.063, 74.387]
  MoveL 6751 to (-67.94, 36.02, -7.81) mm, rotated rx -180 ry 0 rz 90 deg; joints [74.367, -18.772, 89.793, 0, 18.98, 74.367]
  MoveL 6752 to (-69.37, 35.51, -8.22) mm, rotated rx -180 ry 0 rz 90 deg; joints [74.336, -18.77, 89.865, 0, 18.905, 74.336]
  MoveL 6753 to (-70.66, 34.69, -8.63) mm, rotated rx 180 ry 0 rz 90 deg; joints [74.296, -18.764, 89.922, 0, 18.842, 74.296]
  MoveL 6754 to (-71.72, 33.61, -9.03) mm, rotated rx -180 ry 0 rz 90 deg; joints [74.249, -18.754, 89.959, 0, 18.795, 74.249]
  MoveL 6755 to (-72.53, 32.32, -9.44) mm, rotated rx 180 ry 0 rz 90 deg; joints [74.197, -18.739, 89.975, 0, 18.764, 74.197]
  MoveL 6756 to (-73.03, 30.89, -9.84) mm, rotated rx 180 ry 0 rz 90 deg; joints [74.144, -18.719, 89.967, 0, 18.752, 74.144]
  MoveL 6757 to (-73.17, 29.38, -10.25) mm, rotated rx -180 ry 0 rz 90 deg; joints [74.091, -18.694, 89.934, 0, 18.76, 74.091]
  MoveL 6758 to (-73.17, 3.32, -10.25) mm, rotated rx 180 ry 0 rz 90 deg; joints [73.211, -18.581, 89.423, 0, 19.158, 73.211]
  MoveL 6759 to (-73.16, 2.37, -10.25) mm, rotated rx 180 ry 0 rz 90 deg; joints [73.179, -18.577, 89.403, 0, 19.173, 73.179]
  MoveC 6760 to (-72.28, 0.17, -10.25) mm, rotated rx -180 ry 0 rz 90 deg; joints [73.114, -18.553, 89.3, 0, 19.254, 73.114] to (-70.13, -0.83, -10.25) mm, rotated rx 180 ry 0 rz 90 deg; joints [73.102, -18.516, 89.135, 0, 19.381, 73.102]
  MoveC 6761 to (-69.87, -0.82, -10.25) mm, rotated rx -180 ry 0 rz 90 deg; joints [73.105, -18.513, 89.118, 0, 19.395, 73.105] to (-69.61, -0.78, -10.25) mm, rotated rx 180 ry 0 rz 90 deg; joints [73.109, -18.509, 89.102, 0, 19.407, 73.109]
  MoveC 6762 to (-46.55, 4.59, -10.25) mm, rotated rx 180 ry 0 rz 90 deg; joints [73.519, -18.174, 87.65, 0, 20.524, 73.519] to (-23.51, 10.03, -10.25) mm, rotated rx -180 ry 0 rz 90 deg; joints [73.92, -17.817, 86.172, 0, 21.645, 73.92]
  MoveC 6763 to (-22.88, 10.2, -10.25) mm, rotated rx 180 ry 0 rz 90 deg; joints [73.932, -17.807, 86.132, 0, 21.675, 73.932] to (-22.27, 10.41, -10.25) mm, rotated rx 180 ry 0 rz 90 deg; joints [73.945, -17.798, 86.094, 0, 21.704, 73.945]
  MoveC 6764 to (-20.94, 11.84, -10.25) mm, rotated rx 180 ry 0 rz 90 deg; joints [74.004, -17.782, 86.03, 0, 21.752, 74.004] to (-20.54, 13.74, -10.25) mm, rotated rx -180 ry 0 rz 90 deg; joints [74.07, -17.784, 86.04, 0, 21.744, 74.07]
  MoveC 6765 to (-20.66, 14.22, -10.25) mm, rotated rx 180 ry 0 rz 90 deg; joints [74.085, -17.789, 86.057, 0, 21.731, 74.085] to (-20.81, 14.69, -10.25) mm, rotated rx -180 ry 0 rz 90 deg; joints [74.099, -17.794, 86.077, 0, 21.716, 74.099]
  MoveL 6766 to (-26.71, 31.25, -10.25) mm, rotated rx 180 ry 0 rz 90 deg; joints [74.59, -17.973, 86.809, 0, 21.163, 74.59]
  MoveC 6767 to (-27.09, 31.98, -10.25) mm, rotated rx 180 ry 0 rz 90 deg; joints [74.611, -17.982, 86.85, 0, 21.133, 74.611] to (-27.66, 32.59, -10.25) mm, rotated rx 180 ry 0 rz 90 deg; joints [74.626, -17.995, 86.9, 0, 21.094, 74.626]
  MoveC 6768 to (-27.96, 32.82, -10.25) mm, rotated rx -180 ry 0 rz 90 deg; joints [74.631, -18.001, 86.926, 0, 21.075, 74.631] to (-28.28, 33.04, -10.25) mm, rotated rx -180 ry 0 rz 90 deg; joints [74.635, -18.007, 86.952, 0, 21.055, 74.635]
  MoveL 6769 to (-33.64, 36.53, -10.25) mm, rotated rx 180 ry 0 rz 90 deg; joints [74.703, -18.112, 87.388, 0, 20.723, 74.703]
  MoveL 6770 to (-64.4, 56.39, -10.25) mm, rotated rx -180 ry 0 rz 90 deg; joints [75.092, -18.674, 89.845, 0, 18.829, 75.092]
  MoveL 6771 to (-68.7, 59.15, -10.25) mm, rotated rx 180 ry 0 rz 90 deg; joints [75.147, -18.748, 90.184, 0, 18.565, 75.147]
  MoveC 6772 to (-70.58, 59.22, -10.25) mm, rotated rx -180 ry 0 rz 90 deg; joints [75.132, -18.776, 90.31, 0, 18.465, 75.132] to (-72.21, 58.28, -10.25) mm, rotated rx 180 ry 0 rz 90 deg; joints [75.085, -18.796, 90.403, 0, 18.393, 75.085]
  MoveC 6773 to (-72.91, 57.44, -10.25) mm, rotated rx -180 ry 0 rz 90 deg; joints [75.05, -18.803, 90.434, 0, 18.368, 75.05] to (-73.16, 56.39, -10.25) mm, rotated rx 180 ry 0 rz 90 deg; joints [75.012, -18.802, 90.432, 0, 18.37, 75.012]
  MoveL 6774 to (-73.17, 55.91, -10.25) mm, rotated rx 180 ry 0 rz 90 deg; joints [74.996, -18.8, 90.424, 0, 18.376, 74.996]
  MoveL 6775 to (-73.17, 29.38, -10.25) mm, rotated rx -180 ry 0 rz 90 deg; joints [74.091, -18.694, 89.934, 0, 18.76, 74.091]
  MoveL 6776 to (-65.62, 29.38, -10.25) mm, rotated rx 180 ry 0 rz 90 deg; joints [74.164, -18.582, 89.428, 0, 19.154, 74.164]
  MoveL 6777 to (-65.62, 29.38, -7.25) mm, rotated rx -180 ry 0 rz 90 deg; joints [74.164, -18.739, 89.53, 0, 19.209, 74.164]
  Establecer velocidad (1000.0 mm/s)
  MoveL 6778 to (-65.62, 29.38, 10) mm, rotated rx 180 ry 0 rz 90 deg; joints [74.164, -19.641, 90.107, 0, 19.534, 74.164]
  Establecer velocidad (66.7 mm/s)
  MoveL 6779 to (-64.76, 36.02, 10) mm, rotated rx 180 ry 0 rz 90 deg; joints [74.397, -19.656, 90.175, 0, 19.481, 74.397]
  MoveL 6780 to (-64.76, 36.02, -7.25) mm, rotated rx 180 ry 0 rz 90 deg; joints [74.397, -18.754, 89.598, 0, 19.156, 74.397]
  MoveL 6781 to (-66.27, 36.2, -7.66) mm, rotated rx 180 ry 0 rz 90 deg; joints [74.389, -18.756, 89.689, 0, 19.067, 74.389]
  MoveL 6782 to (-67.78, 36.02, -8.06) mm, rotated rx 180 ry 0 rz 90 deg; joints [74.368, -18.757, 89.773, 0, 18.984, 74.368]
  MoveL 6783 to (-69.21, 35.51, -8.47) mm, rotated rx 180 ry 0 rz 90 deg; joints [74.337, -18.755, 89.846, 0, 18.909, 74.337]
  MoveL 6784 to (-70.49, 34.69, -8.87) mm, rotated rx -180 ry 0 rz 90 deg; joints [74.297, -18.749, 89.902, 0, 18.846, 74.297]
  MoveL 6785 to (-71.56, 33.61, -9.28) mm, rotated rx 180 ry 0 rz 90 deg; joints [74.25, -18.739, 89.94, 0, 18.799, 74.25]
  MoveL 6786 to (-72.36, 32.32, -9.69) mm, rotated rx 180 ry 0 rz 90 deg; joints [74.199, -18.724, 89.955, 0, 18.768, 74.199]
  MoveL 6787 to (-72.86, 30.89, -10.09) mm, rotated rx -180 ry 0 rz 90 deg; joints [74.145, -18.704, 89.948, 0, 18.756, 74.145]
  MoveL 6788 to (-73, 29.38, -10.5) mm, rotated rx 180 ry 0 rz 90 deg; joints [74.093, -18.678, 89.915, 0, 18.764, 74.093]
  MoveL 6789 to (-73, 3.32, -10.5) mm, rotated rx -180 ry 0 rz 90 deg; joints [73.212, -18.565, 89.403, 0, 19.162, 73.212]
  MoveL 6790 to (-72.99, 2.37, -10.5) mm, rotated rx -180 ry 0 rz 90 deg; joints [73.181, -18.561, 89.383, 0, 19.178, 73.181]
  MoveC 6791 to (-71.95, 0.17, -10.5) mm, rotated rx 180 ry 0 rz 90 deg; joints [73.117, -18.535, 89.269, 0, 19.266, 73.117] to (-69.65, -0.62, -10.5) mm, rotated rx -180 ry 0 rz 90 deg; joints [73.114, -18.497, 89.099, 0, 19.398, 73.114]
  MoveL 6792 to (-68.91, -0.47, -10.5) mm, rotated rx -180 ry 0 rz 90 deg; joints [73.127, -18.487, 89.052, 0, 19.434, 73.127]
  MoveC 6793 to (-46.06, 4.86, -10.5) mm, rotated rx -180 ry 0 rz 90 deg; joints [73.533, -18.154, 87.613, 0, 20.541, 73.533] to (-23.22, 10.27, -10.5) mm, rotated rx 180 ry 0 rz 90 deg; joints [73.931, -17.8, 86.148, 0, 21.652, 73.931]
  MoveC 6794 to (-22.12, 10.77, -10.5) mm, rotated rx 180 ry 0 rz 90 deg; joints [73.958, -17.784, 86.082, 0, 21.702, 73.958] to (-21.32, 11.66, -10.5) mm, rotated rx -180 ry 0 rz 90 deg; joints [73.995, -17.775, 86.044, 0, 21.73, 73.995]
  MoveC 6795 to (-20.77, 13.13, -10.5) mm, rotated rx 180 ry 0 rz 90 deg; joints [74.048, -17.772, 86.035, 0, 21.738, 74.048] to (-20.98, 14.69, -10.5) mm, rotated rx 180 ry 0 rz 90 deg; joints [74.097, -17.784, 86.08, 0, 21.703, 74.097]
  MoveL 6796 to (-26.82, 31.12, -10.5) mm, rotated rx 180 ry 0 rz 90 deg; joints [74.585, -17.961, 86.806, 0, 21.155, 74.585]
  MoveC 6797 to (-27.32, 32.02, -10.5) mm, rotated rx 180 ry 0 rz 90 deg; joints [74.61, -17.973, 86.858, 0, 21.116, 74.61] to (-28.08, 32.71, -10.5) mm, rotated rx 180 ry 0 rz 90 deg; joints [74.626, -17.989, 86.923, 0, 21.066, 74.626]
  MoveC 6798 to (-48.25, 45.8, -10.5) mm, rotated rx 180 ry 0 rz 90 deg; joints [74.88, -18.373, 88.552, 0, 19.821, 74.88] to (-68.46, 58.83, -10.5) mm, rotated rx -180 ry 0 rz 90 deg; joints [75.139, -18.73, 90.153, 0, 18.578, 75.139]
  MoveC 6799 to (-68.78, 58.99, -10.5) mm, rotated rx 180 ry 0 rz 90 deg; joints [75.141, -18.736, 90.177, 0, 18.559, 75.141] to (-69.13, 59.06, -10.5) mm, rotated rx -180 ry 0 rz 90 deg; joints [75.14, -18.741, 90.202, 0, 18.539, 75.14]
  MoveC 6800 to (-71.13, 58.68, -10.5) mm, rotated rx 180 ry 0 rz 90 deg; joints [75.109, -18.769, 90.329, 0, 18.439, 75.109] to (-72.66, 57.33, -10.5) mm, rotated rx 180 ry 0 rz 90 deg; joints [75.049, -18.785, 90.407, 0, 18.378, 75.049]
  MoveC 6801 to (-72.89, 56.88, -10.5) mm, rotated rx -180 ry 0 rz 90 deg; joints [75.031, -18.787, 90.415, 0, 18.372, 75.031] to (-72.99, 56.39, -10.5) mm, rotated rx -180 ry 0 rz 90 deg; joints [75.013, -18.786, 90.413, 0, 18.374, 75.013]
  MoveL 6802 to (-73, 55.91, -10.5) mm, rotated rx -180 ry 0 rz 90 deg; joints [74.997, -18.785, 90.405, 0, 18.38, 74.997]
  MoveL 6803 to (-73, 29.38, -10.5) mm, rotated rx 180 ry 0 rz 90 deg; joints [74.093, -18.678, 89.915, 0, 18.764, 74.093]
  MoveL 6804 to (-65.45, 29.38, -10.5) mm, rotated rx 180 ry 0 rz 90 deg; joints [74.165, -18.566, 89.409, 0, 19.158, 74.165]
  MoveL 6805 to (-65.45, 29.38, -7.5) mm, rotated rx -180 ry 0 rz 90 deg; joints [74.165, -18.723, 89.511, 0, 19.213, 74.165]
  Establecer velocidad (1000.0 mm/s)
  MoveL 6806 to (-65.45, 29.38, 10) mm, rotated rx 180 ry 0 rz 90 deg; joints [74.165, -19.638, 90.096, 0, 19.542, 74.165]
  Establecer velocidad (66.7 mm/s)
  MoveL 6807 to (-39.92, -32.58, 10) mm, rotated rx 180 ry 0 rz 90 deg; joints [72.363, -18.921, 87.093, 0, 21.828, 72.363]
  MoveL 6808 to (-39.92, -32.58, -7.25) mm, rotated rx -180 ry 0 rz 90 deg; joints [72.363, -18.031, 86.516, 0, 21.515, 72.363]
  MoveL 6809 to (-40.05, -31.07, -7.66) mm, rotated rx -180 ry 0 rz 90 deg; joints [72.411, -18.021, 86.544, 0, 21.477, 72.411]
  MoveL 6810 to (-40.53, -29.63, -8.06) mm, rotated rx -180 ry 0 rz 90 deg; joints [72.453, -18.015, 86.595, 0, 21.421, 72.453]
  MoveL 6811 to (-41.32, -28.33, -8.47) mm, rotated rx 180 ry 0 rz 90 deg; joints [72.487, -18.015, 86.664, 0, 21.351, 72.487]
  MoveL 6812 to (-42.38, -27.24, -8.87) mm, rotated rx -180 ry 0 rz 90 deg; joints [72.512, -18.017, 86.746, 0, 21.271, 72.512]
  MoveL 6813 to (-43.65, -26.41, -9.28) mm, rotated rx 180 ry 0 rz 90 deg; joints [72.526, -18.022, 86.837, 0, 21.184, 72.526]
  MoveL 6814 to (-45.08, -25.89, -9.69) mm, rotated rx 180 ry 0 rz 90 deg; joints [72.528, -18.027, 86.933, 0, 21.094, 72.528]
  MoveL 6815 to (-46.59, -25.69, -10.09) mm, rotated rx 180 ry 0 rz 90 deg; joints [72.519, -18.032, 87.026, 0, 21.006, 72.519]
  MoveL 6816 to (-48.09, -25.86, -10.5) mm, rotated rx -180 ry 0 rz 90 deg; joints [72.498, -18.035, 87.112, 0, 20.923, 72.498]
  MoveL 6817 to (-64.91, -29.34, -10.5) mm, rotated rx -180 ry 0 rz 90 deg; joints [72.207, -18.286, 88.177, 0, 20.109, 72.207]
  MoveL 6818 to (-70.6, -30.54, -10.5) mm, rotated rx 180 ry 0 rz 90 deg; joints [72.106, -18.369, 88.534, 0, 19.835, 72.106]
  MoveC 6819 to (-72.22, -31.46, -10.5) mm, rotated rx 180 ry 0 rz 90 deg; joints [72.058, -18.389, 88.623, 0, 19.766, 72.058] to (-72.97, -33.17, -10.5) mm, rotated rx 180 ry 0 rz 90 deg; joints [71.994, -18.392, 88.636, 0, 19.756, 71.994]
  MoveL 6820 to (-73, -33.64, -10.5) mm, rotated rx 180 ry 0 rz 90 deg; joints [71.978, -18.39, 88.627, 0, 19.763, 71.978]
  MoveL 6821 to (-73, -34.59, -10.5) mm, rotated rx 180 ry 0 rz 90 deg; joints [71.946, -18.385, 88.607, 0, 19.778, 71.946]
  MoveL 6822 to (-73, -68.7, -10.5) mm, rotated rx -180 ry 0 rz 90 deg; joints [70.822, -18.207, 87.836, 0, 20.37, 70.822]
  MoveL 6823 to (-72.99, -69.55, -10.5) mm, rotated rx 180 ry 0 rz 90 deg; joints [70.795, -18.202, 87.816, 0, 20.386, 70.795]
  MoveC 6824 to (-72.07, -71.67, -10.5) mm, rotated rx 180 ry 0 rz 90 deg; joints [70.736, -18.175, 87.704, 0, 20.472, 70.736] to (-69.91, -72.53, -10.5) mm, rotated rx 180 ry 0 rz 90 deg; joints [70.732, -18.136, 87.539, 0, 20.598, 70.732]
  MoveL 6825 to (-38.38, -72.14, -10.5) mm, rotated rx -180 ry 0 rz 90 deg; joints [71.098, -17.614, 85.4, 0, 22.214, 71.098]
  MoveL 6826 to (-36.33, -72.1, -10.5) mm, rotated rx -180 ry 0 rz 90 deg; joints [71.122, -17.578, 85.259, 0, 22.319, 71.122]
  MoveC 6827 to (-34.48, -71.44, -10.5) mm, rotated rx -180 ry 0 rz 90 deg; joints [71.163, -17.55, 85.147, 0, 22.403, 71.163] to (-33.4, -69.78, -10.5) mm, rotated rx 180 ry 0 rz 90 deg; joints [71.228, -17.541, 85.111, 0, 22.43, 71.228]
  MoveL 6828 to (-21.86, -25.25, -10.5) mm, rotated rx -180 ry 0 rz 90 deg; joints [72.786, -17.592, 85.314, 0, 22.278, 72.786]
  MoveC 6829 to (-21.8, -24.95, -10.5) mm, rotated rx -180 ry 0 rz 90 deg; joints [72.796, -17.593, 85.316, 0, 22.276, 72.796] to (-21.76, -24.64, -10.5) mm, rotated rx -180 ry 0 rz 90 deg; joints [72.806, -17.594, 85.321, 0, 22.273, 72.806]
  MoveC 6830 to (-22.57, -22.64, -10.5) mm, rotated rx 180 ry 0 rz 90 deg; joints [72.863, -17.619, 85.42, 0, 22.199, 72.863] to (-24.26, -21.32, -10.5) mm, rotated rx -180 ry 0 rz 90 deg; joints [72.889, -17.656, 85.566, 0, 22.09, 72.889]
  MoveC 6831 to (-24.91, -21.16, -10.5) mm, rotated rx -180 ry 0 rz 90 deg; joints [72.888, -17.668, 85.615, 0, 22.053, 72.888] to (-25.59, -21.2, -10.5) mm, rotated rx 180 ry 0 rz 90 deg; joints [72.879, -17.679, 85.661, 0, 22.019, 72.879]
  MoveL 6832 to (-29.85, -22.08, -10.5) mm, rotated rx 180 ry 0 rz 90 deg; joints [72.808, -17.748, 85.938, 0, 21.81, 72.808]
  MoveL 6833 to (-48.09, -25.86, -10.5) mm, rotated rx -180 ry 0 rz 90 deg; joints [72.498, -18.035, 87.112, 0, 20.923, 72.498]
  MoveL 6834 to (-46.56, -33.25, -10.5) mm, rotated rx 180 ry 0 rz 90 deg; joints [72.272, -17.971, 86.846, 0, 21.124, 72.272]
  MoveL 6835 to (-46.56, -33.25, -7.5) mm, rotated rx -180 ry 0 rz 90 deg; joints [72.272, -18.126, 86.948, 0, 21.178, 72.272]
  Establecer velocidad (1000.0 mm/s)
  MoveL 6836 to (-46.56, -33.25, 10) mm, rotated rx -180 ry 0 rz 90 deg; joints [72.272, -19.03, 87.534, 0, 21.497, 72.272]
  Establecer velocidad (66.7 mm/s)
  MoveL 6837 to (14.97, -63.1, 10) mm, rotated rx -180 ry 0 rz 90 deg; joints [71.951, -17.719, 82.54, 0, 25.179, 71.951]
  MoveL 6838 to (14.97, -63.1, -7.25) mm, rotated rx 180 ry 0 rz 90 deg; joints [71.951, -16.846, 81.961, 0, 24.885, 71.951]
  MoveL 6839 to (14.84, -64.61, -7.66) mm, rotated rx 180 ry 0 rz 90 deg; joints [71.903, -16.818, 81.921, 0, 24.897, 71.903]
  MoveL 6840 to (15.07, -66.11, -8.06) mm, rotated rx 180 ry 0 rz 90 deg; joints [71.858, -16.783, 81.855, 0, 24.928, 71.858]
  MoveL 6841 to (15.63, -67.52, -8.47) mm, rotated rx -180 ry 0 rz 90 deg; joints [71.819, -16.742, 81.767, 0, 24.975, 71.819]
  MoveL 6842 to (16.49, -68.77, -8.87) mm, rotated rx 180 ry 0 rz 90 deg; joints [71.789, -16.696, 81.661, 0, 25.035, 71.789]
  MoveL 6843 to (17.61, -69.81, -9.28) mm, rotated rx -180 ry 0 rz 90 deg; joints [71.768, -16.646, 81.542, 0, 25.104, 71.768]
  MoveL 6844 to (18.93, -70.57, -9.69) mm, rotated rx 180 ry 0 rz 90 deg; joints [71.758, -16.594, 81.415, 0, 25.18, 71.758]
  MoveL 6845 to (20.38, -71.02, -10.09) mm, rotated rx 180 ry 0 rz 90 deg; joints [71.759, -16.542, 81.285, 0, 25.257, 71.759]
  MoveL 6846 to (21.89, -71.1, -10.5) mm, rotated rx -180 ry 0 rz 90 deg; joints [71.772, -16.49, 81.159, 0, 25.331, 71.772]
  MoveC 6847 to (31.92, -70.72, -10.5) mm, rotated rx 180 ry 0 rz 90 deg; joints [71.886, -16.288, 80.437, 0, 25.851, 71.886] to (41.94, -70.27, -10.5) mm, rotated rx -180 ry 0 rz 90 deg; joints [72.001, -16.082, 79.71, 0, 26.372, 72.001]
  MoveC 6848 to (43.51, -68.8, -10.5) mm, rotated rx 180 ry 0 rz 90 deg; joints [72.062, -16.059, 79.63, 0, 26.429, 72.062] to (44.32, -66.81, -10.5) mm, rotated rx -180 ry 0 rz 90 deg; joints [72.132, -16.055, 79.617, 0, 26.438, 72.132]
  MoveC 6849 to (44.55, -65.08, -10.5) mm, rotated rx -180 ry 0 rz 90 deg; joints [72.188, -16.062, 79.641, 0, 26.421, 72.188] to (44.07, -63.41, -10.5) mm, rotated rx 180 ry 0 rz 90 deg; joints [72.235, -16.084, 79.717, 0, 26.367, 72.235]
  MoveC 6850 to (34.2, -51.34, -10.5) mm, rotated rx -180 ry 0 rz 90 deg; joints [72.512, -16.369, 80.726, 0, 25.643, 72.512] to (24.21, -39.38, -10.5) mm, rotated rx -180 ry 0 rz 90 deg; joints [72.79, -16.647, 81.726, 0, 24.92, 72.79]
  MoveC 6851 to (23.77, -38.87, -10.5) mm, rotated rx 180 ry 0 rz 90 deg; joints [72.802, -16.659, 81.77, 0, 24.889, 72.802] to (23.32, -38.38, -10.5) mm, rotated rx 180 ry 0 rz 90 deg; joints [72.813, -16.671, 81.814, 0, 24.857, 72.813]
  MoveL 6852 to (13.74, -30.52, -10.5) mm, rotated rx -180 ry 0 rz 90 deg; joints [72.968, -16.906, 82.68, 0, 24.226, 72.968]
  MoveL 6853 to (13.27, -30.16, -10.5) mm, rotated rx 180 ry 0 rz 90 deg; joints [72.975, -16.917, 82.721, 0, 24.196, 72.975]
  MoveC 6854 to (11.08, -29.76, -10.5) mm, rotated rx -180 ry 0 rz 90 deg; joints [72.967, -16.961, 82.887, 0, 24.074, 72.967] to (9, -30.56, -10.5) mm, rotated rx -180 ry 0 rz 90 deg; joints [72.921, -16.996, 83.018, 0, 23.978, 72.921]
  MoveC 6855 to (8.46, -31.12, -10.5) mm, rotated rx -180 ry 0 rz 90 deg; joints [72.897, -17.003, 83.045, 0, 23.959, 72.897] to (8.14, -31.84, -10.5) mm, rotated rx -180 ry 0 rz 90 deg; joints [72.872, -17.005, 83.052, 0, 23.953, 72.872]
  MoveL 6856 to (-1.52, -67.56, -10.5) mm, rotated rx 180 ry 0 rz 90 deg; joints [71.64, -16.972, 82.926, 0, 24.046, 71.64]
  MoveC 6857 to (-1.62, -68.25, -10.5) mm, rotated rx 180 ry 0 rz 90 deg; joints [71.617, -16.969, 82.917, 0, 24.053, 71.617] to (-1.56, -68.94, -10.5) mm, rotated rx 180 ry 0 rz 90 deg; joints [71.596, -16.964, 82.896, 0, 24.068, 71.596]
  MoveC 6858 to (-0.36, -70.91, -10.5) mm, rotated rx -180 ry 0 rz 90 deg; joints [71.546, -16.928, 82.764, 0, 24.165, 71.546] to (1.83, -71.66, -10.5) mm, rotated rx -180 ry 0 rz 90 deg; joints [71.546, -16.882, 82.59, 0, 24.292, 71.546]
  MoveC 6859 to (11.86, -71.41, -10.5) mm, rotated rx -180 ry 0 rz 90 deg; joints [71.658, -16.688, 81.877, 0, 24.811, 71.658] to (21.89, -71.1, -10.5) mm, rotated rx -180 ry 0 rz 90 deg; joints [71.772, -16.49, 81.159, 0, 25.331, 71.772]
  MoveL 6860 to (21.63, -63.56, -10.5) mm, rotated rx -180 ry 0 rz 90 deg; joints [72.005, -16.545, 81.357, 0, 25.188, 72.005]
  MoveL 6861 to (21.63, -63.56, -7.5) mm, rotated rx -180 ry 0 rz 90 deg; joints [72.005, -16.697, 81.46, 0, 25.237, 72.005]
  Establecer velocidad (1000.0 mm/s)
  MoveL 6862 to (21.63, -63.56, 10) mm, rotated rx 180 ry 0 rz 90 deg; joints [72.005, -17.582, 82.048, 0, 25.534, 72.005]
  Establecer velocidad (66.7 mm/s)
  MoveL 6863 to (35.03, 18.14, 10) mm, rotated rx 180 ry 0 rz 90 deg; joints [74.715, -17.805, 82.849, 0, 24.956, 74.715]
  MoveL 6864 to (35.03, 18.14, -7.25) mm, rotated rx -180 ry 0 rz 90 deg; joints [74.715, -16.93, 82.27, 0, 24.66, 74.715]
  MoveL 6865 to (35.21, 19.65, -7.66) mm, rotated rx -180 ry 0 rz 90 deg; joints [74.765, -16.914, 82.273, 0, 24.641, 74.765]
  MoveL 6866 to (35.03, 21.16, -8.06) mm, rotated rx -180 ry 0 rz 90 deg; joints [74.811, -16.905, 82.302, 0, 24.603, 74.811]
  MoveL 6867 to (34.51, 22.59, -8.47) mm, rotated rx -180 ry 0 rz 90 deg; joints [74.853, -16.902, 82.354, 0, 24.548, 74.853]
  MoveL 6868 to (33.7, 23.87, -8.87) mm, rotated rx 180 ry 0 rz 90 deg; joints [74.887, -16.905, 82.425, 0, 24.48, 74.887]
  MoveL 6869 to (32.62, 24.94, -9.28) mm, rotated rx 180 ry 0 rz 90 deg; joints [74.912, -16.911, 82.511, 0, 24.4, 74.912]
  MoveL 6870 to (31.33, 25.74, -9.69) mm, rotated rx 180 ry 0 rz 90 deg; joints [74.926, -16.92, 82.606, 0, 24.314, 74.926]
  MoveL 6871 to (29.89, 26.24, -10.09) mm, rotated rx 180 ry 0 rz 90 deg; joints [74.93, -16.93, 82.706, 0, 24.224, 74.93]
  MoveL 6872 to (28.38, 26.38, -10.5) mm, rotated rx -180 ry 0 rz 90 deg; joints [74.921, -16.939, 82.805, 0, 24.135, 74.921]
  MoveC 6873 to (21.06, 26.35, -10.5) mm, rotated rx 180 ry 0 rz 90 deg; joints [74.857, -17.08, 83.333, 0, 23.747, 74.857] to (13.74, 26.29, -10.5) mm, rotated rx -180 ry 0 rz 90 deg; joints [74.791, -17.218, 83.857, 0, 23.361, 74.791]
  MoveC 6874 to (11.07, 25.08, -10.5) mm, rotated rx 180 ry 0 rz 90 deg; joints [74.728, -17.262, 84.025, 0, 23.237, 74.728] to (10.25, 22.27, -10.5) mm, rotated rx 180 ry 0 rz 90 deg; joints [74.63, -17.263, 84.028, 0, 23.234, 74.63]
  MoveL 6875 to (10.44, 21.73, -10.5) mm, rotated rx -180 ry 0 rz 90 deg; joints [74.614, -17.256, 84.004, 0, 23.252, 74.614]
  MoveL 6876 to (14.08, 11.85, -10.5) mm, rotated rx -180 ry 0 rz 90 deg; joints [74.327, -17.137, 83.548, 0, 23.589, 74.327]
  MoveL 6877 to (14.4, 11, -10.5) mm, rotated rx -180 ry 0 rz 90 deg; joints [74.303, -17.126, 83.507, 0, 23.619, 74.303]
  MoveC 6878 to (14.81, 10.27, -10.5) mm, rotated rx 180 ry 0 rz 90 deg; joints [74.283, -17.115, 83.464, 0, 23.651, 74.283] to (15.39, 9.69, -10.5) mm, rotated rx -180 ry 0 rz 90 deg; joints [74.269, -17.1, 83.41, 0, 23.691, 74.269]
  MoveL 6879 to (16.29, 9, -10.5) mm, rotated rx 180 ry 0 rz 90 deg; joints [74.256, -17.08, 83.331, 0, 23.748, 74.256]
  MoveL 6880 to (28.33, 0.01, -10.5) mm, rotated rx -180 ry 0 rz 90 deg; joints [74.077, -16.797, 82.278, 0, 24.52, 74.077]
  MoveC 6881 to (28.91, -0.32, -10.5) mm, rotated rx 180 ry 0 rz 90 deg; joints [74.072, -16.784, 82.229, 0, 24.555, 74.072] to (29.55, -0.49, -10.5) mm, rotated rx -180 ry 0 rz 90 deg; joints [74.072, -16.77, 82.179, 0, 24.591, 74.072]
  MoveC 6882 to (31.68, -0.19, -10.5) mm, rotated rx 180 ry 0 rz 90 deg; joints [74.101, -16.73, 82.03, 0, 24.7, 74.101] to (33.33, 1.18, -10.5) mm, rotated rx -180 ry 0 rz 90 deg; joints [74.16, -16.705, 81.938, 0, 24.767, 74.16]
  MoveL 6883 to (45.24, 18.48, -10.5) mm, rotated rx 180 ry 0 rz 90 deg; joints [74.814, -16.562, 81.418, 0, 25.144, 74.814]
  MoveL 6884 to (46.28, 20.04, -10.5) mm, rotated rx -180 ry 0 rz 90 deg; joints [74.873, -16.549, 81.373, 0, 25.177, 74.873]
  MoveC 6885 to (46.04, 23.37, -10.5) mm, rotated rx -180 ry 0 rz 90 deg; joints [74.977, -16.572, 81.456, 0, 25.116, 74.977] to (44.07, 26.06, -10.5) mm, rotated rx 180 ry 0 rz 90 deg; joints [75.046, -16.627, 81.654, 0, 24.973, 75.046]
  MoveC 6886 to (43.56, 26.25, -10.5) mm, rotated rx 180 ry 0 rz 90 deg; joints [75.047, -16.638, 81.695, 0, 24.943, 75.047] to (43.02, 26.32, -10.5) mm, rotated rx 180 ry 0 rz 90 deg; joints [75.045, -16.649, 81.736, 0, 24.913, 75.045]
  MoveC 6887 to (35.7, 26.36, -10.5) mm, rotated rx -180 ry 0 rz 90 deg; joints [74.984, -16.796, 82.272, 0, 24.523, 74.984] to (28.38, 26.38, -10.5) mm, rotated rx -180 ry 0 rz 90 deg; joints [74.921, -16.939, 82.805, 0, 24.135, 74.921]
  MoveL 6888 to (28.39, 18.83, -10.5) mm, rotated rx 180 ry 0 rz 90 deg; joints [74.679, -16.899, 82.656, 0, 24.244, 74.679]
  MoveL 6889 to (28.39, 18.83, -7.5) mm, rotated rx 180 ry 0 rz 90 deg; joints [74.679, -17.052, 82.758, 0, 24.294, 74.679]
  Establecer velocidad (1000.0 mm/s)
  MoveL 6890 to (28.39, 18.83, 10) mm, rotated rx 180 ry 0 rz 90 deg; joints [74.679, -17.941, 83.345, 0, 24.596, 74.679]
  Establecer velocidad (66.7 mm/s)
  MoveL 6891 to (4.27, 58.51, 10) mm, rotated rx 180 ry 0 rz 90 deg; joints [75.76, -18.599, 85.823, 0, 22.776, 75.76]
  MoveL 6892 to (4.27, 58.51, -7.25) mm, rotated rx 180 ry 0 rz 90 deg; joints [75.76, -17.714, 85.246, 0, 22.468, 75.76]
  MoveL 6893 to (5.67, 57.92, -7.66) mm, rotated rx 180 ry 0 rz 90 deg; joints [75.752, -17.665, 85.122, 0, 22.543, 75.752]
  MoveL 6894 to (7.17, 57.69, -8.06) mm, rotated rx -180 ry 0 rz 90 deg; joints [75.757, -17.616, 84.998, 0, 22.619, 75.757]
  MoveL 6895 to (8.69, 57.79, -8.47) mm, rotated rx -180 ry 0 rz 90 deg; joints [75.773, -17.568, 84.878, 0, 22.69, 75.773]
  MoveL 6896 to (10.14, 58.23, -8.87) mm, rotated rx -180 ry 0 rz 90 deg; joints [75.8, -17.523, 84.768, 0, 22.755, 75.8]
  MoveL 6897 to (11.47, 58.98, -9.28) mm, rotated rx 180 ry 0 rz 90 deg; joints [75.835, -17.481, 84.674, 0, 22.808, 75.835]
  MoveL 6898 to (12.59, 60, -9.69) mm, rotated rx 180 ry 0 rz 90 deg; joints [75.878, -17.445, 84.598, 0, 22.846, 75.878]
  MoveL 6899 to (13.46, 61.25, -10.09) mm, rotated rx -180 ry 0 rz 90 deg; joints [75.926, -17.414, 84.544, 0, 22.869, 75.926]
  MoveL 6900 to (14, 62.66, -10.5) mm, rotated rx -180 ry 0 rz 90 deg; joints [75.976, -17.389, 84.517, 0, 22.872, 75.976]
  MoveL 6901 to (16.36, 71.03, -10.5) mm, rotated rx -180 ry 0 rz 90 deg; joints [76.269, -17.384, 84.496, 0, 22.888, 76.269]
  MoveC 6902 to (-1.03, 71.54, -10.5) mm, rotated rx -180 ry 0 rz 90 deg; joints [76.146, -17.699, 85.741, 0, 21.959, 76.146] to (-18.42, 71.94, -10.5) mm, rotated rx 180 ry 0 rz 90 deg; joints [76.016, -18, 86.966, 0, 21.033, 76.016]
  MoveC 6903 to (-20.71, 69.13, -10.5) mm, rotated rx 180 ry 0 rz 90 deg; joints [75.903, -18.026, 87.076, 0, 20.95, 75.903] to (-20.41, 65.52, -10.5) mm, rotated rx 180 ry 0 rz 90 deg; joints [75.785, -18.006, 86.992, 0, 21.014, 75.785]
  MoveL 6904 to (-6.81, 56.73, -10.5) mm, rotated rx 180 ry 0 rz 90 deg; joints [75.608, -17.735, 85.885, 0, 21.85, 75.608]
  MoveC 6905 to (-6.48, 56.59, -10.5) mm, rotated rx 180 ry 0 rz 90 deg; joints [75.606, -17.729, 85.86, 0, 21.869, 75.606] to (-6.12, 56.56, -10.5) mm, rotated rx 180 ry 0 rz 90 deg; joints [75.608, -17.722, 85.834, 0, 21.889, 75.608]
  MoveC 6906 to (12.83, 58.18, -10.5) mm, rotated rx -180 ry 0 rz 90 deg; joints [75.82, -17.39, 84.52, 0, 22.87, 75.82] to (31.75, 60.22, -10.5) mm, rotated rx 180 ry 0 rz 90 deg; joints [76.041, -17.044, 83.196, 0, 23.848, 76.041]
  MoveC 6907 to (41.44, 61.47, -10.5) mm, rotated rx 180 ry 0 rz 90 deg; joints [76.159, -16.861, 82.513, 0, 24.348, 76.159] to (51.1, 62.95, -10.5) mm, rotated rx 180 ry 0 rz 90 deg; joints [76.282, -16.675, 81.83, 0, 24.845, 76.282]
  MoveL 6908 to (51.1, 69.19, -10.5) mm, rotated rx 180 ry 0 rz 90 deg; joints [76.483, -16.706, 81.941, 0, 24.764, 76.483]
  MoveC 6909 to (36.7, 70.19, -10.5) mm, rotated rx 180 ry 0 rz 90 deg; joints [76.403, -16.995, 83.014, 0, 23.981, 76.403] to (22.27, 70.84, -10.5) mm, rotated rx -180 ry 0 rz 90 deg; joints [76.31, -17.273, 84.069, 0, 23.204, 76.31]
  MoveC 6910 to (19.32, 70.93, -10.5) mm, rotated rx 180 ry 0 rz 90 deg; joints [76.29, -17.329, 84.283, 0, 23.046, 76.29] to (16.36, 71.03, -10.5) mm, rotated rx 180 ry 0 rz 90 deg; joints [76.269, -17.384, 84.496, 0, 22.888, 76.269]
  MoveL 6911 to (16.12, 63.48, -10.5) mm, rotated rx 180 ry 0 rz 90 deg; joints [76.021, -17.354, 84.38, 0, 22.974, 76.021]
  MoveL 6912 to (16.12, 63.48, -7.5) mm, rotated rx -180 ry 0 rz 90 deg; joints [76.021, -17.508, 84.482, 0, 23.025, 76.021]
  Establecer velocidad (1000.0 mm/s)
  MoveL 6913 to (16.12, 63.48, 10) mm, rotated rx 180 ry 0 rz 90 deg; joints [76.021, -18.402, 85.068, 0, 23.334, 76.021]
  Establecer velocidad (66.7 mm/s)
  MoveL 6914 to (-0.24, 59.47, 10) mm, rotated rx 180 ry 0 rz 90 deg; joints [75.754, -18.685, 86.159, 0, 22.526, 75.754]
  MoveL 6915 to (-0.24, 59.47, -7.5) mm, rotated rx 180 ry 0 rz 90 deg; joints [75.754, -17.786, 85.574, 0, 22.212, 75.754]
  MoveL 6916 to (0.95, 58.53, -7.91) mm, rotated rx -180 ry 0 rz 90 deg; joints [75.733, -17.74, 85.459, 0, 22.281, 75.733]
  MoveL 6917 to (2.33, 57.9, -8.31) mm, rotated rx 180 ry 0 rz 90 deg; joints [75.724, -17.691, 85.336, 0, 22.355, 75.724]
  MoveL 6918 to (3.82, 57.59, -8.72) mm, rotated rx 180 ry 0 rz 90 deg; joints [75.726, -17.642, 85.211, 0, 22.431, 75.726]
  MoveL 6919 to (5.34, 57.61, -9.13) mm, rotated rx -180 ry 0 rz 90 deg; joints [75.74, -17.594, 85.09, 0, 22.504, 75.74]
  MoveL 6920 to (6.81, 57.98, -9.53) mm, rotated rx 180 ry 0 rz 90 deg; joints [75.764, -17.549, 84.978, 0, 22.57, 75.764]
  MoveL 6921 to (8.17, 58.66, -9.94) mm, rotated rx 180 ry 0 rz 90 deg; joints [75.797, -17.506, 84.88, 0, 22.626, 75.797]
  MoveL 6922 to (9.35, 59.62, -10.34) mm, rotated rx 180 ry 0 rz 90 deg; joints [75.839, -17.468, 84.8, 0, 22.669, 75.839]
  MoveL 6923 to (10.26, 60.84, -10.75) mm, rotated rx 180 ry 0 rz 90 deg; joints [75.886, -17.437, 84.743, 0, 22.693, 75.886]
  MoveL 6924 to (16.36, 70.82, -10.75) mm, rotated rx -180 ry 0 rz 90 deg; joints [76.262, -17.37, 84.484, 0, 22.886, 76.262]
  MoveC 6925 to (-0.72, 71.33, -10.75) mm, rotated rx 180 ry 0 rz 90 deg; joints [76.141, -17.68, 85.707, 0, 21.973, 76.141] to (-17.8, 71.74, -10.75) mm, rotated rx -180 ry 0 rz 90 deg; joints [76.014, -17.976, 86.911, 0, 21.064, 76.014]
  MoveC 6926 to (-20.06, 68.96, -10.75) mm, rotated rx 180 ry 0 rz 90 deg; joints [75.903, -18.002, 87.02, 0, 20.982, 75.903] to (-19.77, 65.39, -10.75) mm, rotated rx 180 ry 0 rz 90 deg; joints [75.786, -17.982, 86.937, 0, 21.045, 75.786]
  MoveL 6927 to (-8.05, 57.82, -10.75) mm, rotated rx -180 ry 0 rz 90 deg; joints [75.634, -17.749, 85.984, 0, 21.765, 75.634]
  MoveL 6928 to (-6.57, 56.86, -10.75) mm, rotated rx 180 ry 0 rz 90 deg; joints [75.614, -17.719, 85.863, 0, 21.856, 75.614]
  MoveL 6929 to (-6.22, 56.69, -10.75) mm, rotated rx -180 ry 0 rz 90 deg; joints [75.612, -17.712, 85.835, 0, 21.877, 75.612]
  MoveL 6930 to (-6.16, 56.68, -10.75) mm, rotated rx 180 ry 0 rz 90 deg; joints [75.612, -17.711, 85.83, 0, 21.881, 75.612]
  MoveC 6931 to (11.25, 58.19, -10.75) mm, rotated rx 180 ry 0 rz 90 deg; joints [75.808, -17.406, 84.625, 0, 22.782, 75.808] to (28.63, 60.04, -10.75) mm, rotated rx -180 ry 0 rz 90 deg; joints [76.01, -17.09, 83.41, 0, 23.68, 76.01]
  MoveC 6932 to (38.45, 61.29, -10.75) mm, rotated rx -180 ry 0 rz 90 deg; joints [76.129, -16.906, 82.719, 0, 24.187, 76.129] to (48.25, 62.75, -10.75) mm, rotated rx -180 ry 0 rz 90 deg; joints [76.254, -16.719, 82.028, 0, 24.691, 76.254]
  MoveL 6933 to (48.25, 69.13, -10.75) mm, rotated rx -180 ry 0 rz 90 deg; joints [76.459, -16.75, 82.142, 0, 24.608, 76.459]
  MoveC 6934 to (34.23, 70.07, -10.75) mm, rotated rx -180 ry 0 rz 90 deg; joints [76.38, -17.03, 83.183, 0, 23.847, 76.38] to (20.2, 70.69, -10.75) mm, rotated rx 180 ry 0 rz 90 deg; joints [76.289, -17.299, 84.207, 0, 23.092, 76.289]
  MoveC 6935 to (18.28, 70.76, -10.75) mm, rotated rx 180 ry 0 rz 90 deg; joints [76.276, -17.335, 84.346, 0, 22.989, 76.276] to (16.36, 70.82, -10.75) mm, rotated rx 180 ry 0 rz 90 deg; joints [76.262, -17.37, 84.484, 0, 22.886, 76.262]
  MoveL 6936 to (16.11, 63.27, -10.75) mm, rotated rx -180 ry 0 rz 90 deg; joints [76.014, -17.34, 84.369, 0, 22.972, 76.014]
  MoveL 6937 to (16.11, 63.27, -7.75) mm, rotated rx 180 ry 0 rz 90 deg; joints [76.014, -17.494, 84.471, 0, 23.023, 76.014]
  Establecer velocidad (1000.0 mm/s)
  MoveL 6938 to (16.11, 63.27, 10) mm, rotated rx 180 ry 0 rz 90 deg; joints [76.014, -18.402, 85.065, 0, 23.337, 76.014]
  Establecer velocidad (66.7 mm/s)
  MoveL 6939 to (35.05, 17.9, 10) mm, rotated rx 180 ry 0 rz 90 deg; joints [74.708, -17.803, 82.842, 0, 24.961, 74.708]
  MoveL 6940 to (35.05, 17.9, -7.5) mm, rotated rx -180 ry 0 rz 90 deg; joints [74.708, -16.916, 82.255, 0, 24.661, 74.708]
  MoveL 6941 to (35.24, 19.4, -7.91) mm, rotated rx 180 ry 0 rz 90 deg; joints [74.757, -16.899, 82.257, 0, 24.642, 74.757]
  MoveL 6942 to (35.06, 20.91, -8.31) mm, rotated rx 180 ry 0 rz 90 deg; joints [74.804, -16.89, 82.287, 0, 24.604, 74.804]
  MoveL 6943 to (34.55, 22.34, -8.72) mm, rotated rx -180 ry 0 rz 90 deg; joints [74.845, -16.888, 82.338, 0, 24.549, 74.845]
  MoveL 6944 to (33.73, 23.62, -9.13) mm, rotated rx -180 ry 0 rz 90 deg; joints [74.879, -16.89, 82.409, 0, 24.481, 74.879]
  MoveL 6945 to (32.65, 24.7, -9.53) mm, rotated rx -180 ry 0 rz 90 deg; joints [74.904, -16.896, 82.495, 0, 24.402, 74.904]
  MoveL 6946 to (31.36, 25.5, -9.94) mm, rotated rx 180 ry 0 rz 90 deg; joints [74.919, -16.905, 82.59, 0, 24.315, 74.919]
  MoveL 6947 to (29.93, 26, -10.34) mm, rotated rx -180 ry 0 rz 90 deg; joints [74.922, -16.915, 82.69, 0, 24.225, 74.922]
  MoveL 6948 to (28.42, 26.14, -10.75) mm, rotated rx 180 ry 0 rz 90 deg; joints [74.914, -16.925, 82.789, 0, 24.136, 74.914]
  MoveC 6949 to (21.03, 26.13, -10.75) mm, rotated rx -180 ry 0 rz 90 deg; joints [74.849, -17.067, 83.322, 0, 23.745, 74.849] to (13.65, 26.06, -10.75) mm, rotated rx -180 ry 0 rz 90 deg; joints [74.782, -17.206, 83.851, 0, 23.355, 74.782]
  MoveC 6950 to (11.31, 24.81, -10.75) mm, rotated rx -180 ry 0 rz 90 deg; joints [74.721, -17.243, 83.994, 0, 23.249, 74.721] to (10.53, 22.27, -10.75) mm, rotated rx 180 ry 0 rz 90 deg; joints [74.632, -17.245, 84, 0, 23.245, 74.632]
  MoveL 6951 to (10.67, 21.79, -10.75) mm, rotated rx -180 ry 0 rz 90 deg; joints [74.618, -17.24, 83.98, 0, 23.259, 74.618]
  MoveL 6952 to (14.56, 11.22, -10.75) mm, rotated rx 180 ry 0 rz 90 deg; joints [74.311, -17.112, 83.492, 0, 23.62, 74.311]
  MoveC 6953 to (14.98, 10.45, -10.75) mm, rotated rx 180 ry 0 rz 90 deg; joints [74.29, -17.1, 83.446, 0, 23.653, 74.29] to (15.6, 9.82, -10.75) mm, rotated rx 180 ry 0 rz 90 deg; joints [74.276, -17.084, 83.389, 0, 23.695, 74.276]
  MoveL 6954 to (16.58, 9.08, -10.75) mm, rotated rx -180 ry 0 rz 90 deg; joints [74.261, -17.062, 83.303, 0, 23.758, 74.261]
  MoveL 6955 to (28.3, 0.36, -10.75) mm, rotated rx 180 ry 0 rz 90 deg; joints [74.088, -16.787, 82.279, 0, 24.508, 74.088]
  MoveC 6956 to (29.02, -0.03, -10.75) mm, rotated rx 180 ry 0 rz 90 deg; joints [74.082, -16.771, 82.218, 0, 24.553, 74.082] to (29.83, -0.19, -10.75) mm, rotated rx 180 ry 0 rz 90 deg; joints [74.084, -16.754, 82.156, 0, 24.598, 74.084]
  MoveC 6957 to (31.73, 0.19, -10.75) mm, rotated rx 180 ry 0 rz 90 deg; joints [74.114, -16.719, 82.026, 0, 24.692, 74.114] to (33.22, 1.42, -10.75) mm, rotated rx -180 ry 0 rz 90 deg; joints [74.166, -16.696, 81.943, 0, 24.753, 74.166]
  MoveL 6958 to (45.01, 18.62, -10.75) mm, rotated rx 180 ry 0 rz 90 deg; joints [74.817, -16.555, 81.429, 0, 25.126, 74.817]
  MoveL 6959 to (45.82, 19.9, -10.75) mm, rotated rx 180 ry 0 rz 90 deg; joints [74.865, -16.545, 81.395, 0, 25.15, 74.865]
  MoveC 6960 to (45.46, 23.38, -10.75) mm, rotated rx 180 ry 0 rz 90 deg; joints [74.972, -16.572, 81.49, 0, 25.081, 74.972] to (43.19, 26.03, -10.75) mm, rotated rx 180 ry 0 rz 90 deg; joints [75.037, -16.632, 81.709, 0, 24.922, 75.037]
  MoveC 6961 to (35.81, 26.11, -10.75) mm, rotated rx -180 ry 0 rz 90 deg; joints [74.977, -16.78, 82.251, 0, 24.528, 74.977] to (28.42, 26.14, -10.75) mm, rotated rx 180 ry 0 rz 90 deg; joints [74.914, -16.925, 82.789, 0, 24.136, 74.914]
  MoveL 6962 to (28.41, 18.59, -10.75) mm, rotated rx 180 ry 0 rz 90 deg; joints [74.672, -16.885, 82.641, 0, 24.244, 74.672]
  MoveL 6963 to (28.41, 18.59, -7.75) mm, rotated rx 180 ry 0 rz 90 deg; joints [74.672, -17.037, 82.743, 0, 24.295, 74.672]
  Establecer velocidad (1000.0 mm/s)
  MoveL 6964 to (28.41, 18.59, 10) mm, rotated rx 180 ry 0 rz 90 deg; joints [74.672, -17.939, 83.338, 0, 24.601, 74.672]
  Establecer velocidad (66.7 mm/s)
  MoveL 6965 to (14.73, -62.89, 10) mm, rotated rx -180 ry 0 rz 90 deg; joints [71.956, -17.725, 82.562, 0, 25.163, 71.956]
  MoveL 6966 to (14.73, -62.89, -7.5) mm, rotated rx 180 ry 0 rz 90 deg; joints [71.956, -16.839, 81.974, 0, 24.865, 71.956]
  MoveL 6967 to (14.6, -64.4, -7.91) mm, rotated rx 180 ry 0 rz 90 deg; joints [71.907, -16.811, 81.934, 0, 24.877, 71.907]
  MoveL 6968 to (14.84, -65.9, -8.31) mm, rotated rx 180 ry 0 rz 90 deg; joints [71.862, -16.776, 81.868, 0, 24.908, 71.862]
  MoveL 6969 to (15.4, -67.31, -8.72) mm, rotated rx -180 ry 0 rz 90 deg; joints [71.824, -16.735, 81.78, 0, 24.955, 71.824]
  MoveL 6970 to (16.27, -68.56, -9.13) mm, rotated rx -180 ry 0 rz 90 deg; joints [71.793, -16.689, 81.674, 0, 25.015, 71.793]
  MoveL 6971 to (17.38, -69.59, -9.53) mm, rotated rx 180 ry 0 rz 90 deg; joints [71.773, -16.64, 81.555, 0, 25.085, 71.773]
  MoveL 6972 to (18.7, -70.35, -9.94) mm, rotated rx -180 ry 0 rz 90 deg; joints [71.763, -16.588, 81.428, 0, 25.16, 71.763]
  MoveL 6973 to (20.15, -70.8, -10.34) mm, rotated rx 180 ry 0 rz 90 deg; joints [71.763, -16.535, 81.298, 0, 25.237, 71.763]
  MoveL 6974 to (21.67, -70.88, -10.75) mm, rotated rx 180 ry 0 rz 90 deg; joints [71.776, -16.484, 81.172, 0, 25.312, 71.776]
  MoveC 6975 to (31.56, -70.49, -10.75) mm, rotated rx 180 ry 0 rz 90 deg; joints [71.89, -16.284, 80.46, 0, 25.824, 71.89] to (41.46, -70.02, -10.75) mm, rotated rx 180 ry 0 rz 90 deg; joints [72.004, -16.081, 79.744, 0, 26.338, 72.004]
  MoveC 6976 to (43.65, -67.12, -10.75) mm, rotated rx -180 ry 0 rz 90 deg; joints [72.116, -16.055, 79.651, 0, 26.404, 72.116] to (43.78, -63.49, -10.75) mm, rotated rx -180 ry 0 rz 90 deg; joints [72.229, -16.077, 79.727, 0, 26.349, 72.229]
  MoveC 6977 to (33.91, -51.38, -10.75) mm, rotated rx 180 ry 0 rz 90 deg; joints [72.508, -16.362, 80.737, 0, 25.625, 72.508] to (23.93, -39.38, -10.75) mm, rotated rx -180 ry 0 rz 90 deg; joints [72.787, -16.64, 81.738, 0, 24.901, 72.787]
  MoveC 6978 to (23.47, -38.86, -10.75) mm, rotated rx -180 ry 0 rz 90 deg; joints [72.799, -16.652, 81.783, 0, 24.869, 72.799] to (22.99, -38.38, -10.75) mm, rotated rx -180 ry 0 rz 90 deg; joints [72.81, -16.665, 81.829, 0, 24.836, 72.81]
  MoveL 6979 to (13.88, -30.9, -10.75) mm, rotated rx 180 ry 0 rz 90 deg; joints [72.958, -16.888, 82.653, 0, 24.235, 72.958]
  MoveC 6980 to (10.97, -30.1, -10.75) mm, rotated rx 180 ry 0 rz 90 deg; joints [72.955, -16.949, 82.879, 0, 24.07, 72.955] to (8.44, -31.75, -10.75) mm, rotated rx -180 ry 0 rz 90 deg; joints [72.877, -16.988, 83.024, 0, 23.963, 72.877]
  MoveL 6981 to (8.14, -32.69, -10.75) mm, rotated rx 180 ry 0 rz 90 deg; joints [72.844, -16.988, 83.024, 0, 23.963, 72.844]
  MoveL 6982 to (-1.09, -66.81, -10.75) mm, rotated rx -180 ry 0 rz 90 deg; joints [71.668, -16.956, 82.904, 0, 24.051, 71.668]
  MoveL 6983 to (-1.34, -67.76, -10.75) mm, rotated rx -180 ry 0 rz 90 deg; joints [71.636, -16.954, 82.899, 0, 24.055, 71.636]
  MoveC 6984 to (-0.53, -70.29, -10.75) mm, rotated rx 180 ry 0 rz 90 deg; joints [71.564, -16.923, 82.782, 0, 24.141, 71.564] to (1.87, -71.43, -10.75) mm, rotated rx 180 ry 0 rz 90 deg; joints [71.553, -16.87, 82.584, 0, 24.286, 71.553]
  MoveL 6985 to (2.37, -71.45, -10.75) mm, rotated rx 180 ry 0 rz 90 deg; joints [71.558, -16.86, 82.548, 0, 24.312, 71.558]
  MoveC 6986 to (12.02, -71.2, -10.75) mm, rotated rx 180 ry 0 rz 90 deg; joints [71.667, -16.674, 81.862, 0, 24.812, 71.667] to (21.67, -70.88, -10.75) mm, rotated rx 180 ry 0 rz 90 deg; joints [71.776, -16.484, 81.172, 0, 25.312, 71.776]
  MoveL 6987 to (21.39, -63.33, -10.75) mm, rotated rx -180 ry 0 rz 90 deg; joints [72.009, -16.539, 81.371, 0, 25.168, 72.009]
  MoveL 6988 to (21.39, -63.33, -7.75) mm, rotated rx -180 ry 0 rz 90 deg; joints [72.009, -16.691, 81.474, 0, 25.217, 72.009]
  Establecer velocidad (1000.0 mm/s)
  MoveL 6989 to (21.39, -63.33, 10) mm, rotated rx 180 ry 0 rz 90 deg; joints [72.009, -17.588, 82.07, 0, 25.518, 72.009]
  Establecer velocidad (66.7 mm/s)
  MoveL 6990 to (-37.45, -51.98, 10) mm, rotated rx 180 ry 0 rz 90 deg; joints [71.758, -18.769, 86.49, 0, 22.279, 71.758]
  MoveL 6991 to (-37.45, -51.98, -7.5) mm, rotated rx 180 ry 0 rz 90 deg; joints [71.758, -17.869, 85.905, 0, 21.964, 71.758]
  MoveL 6992 to (-36.04, -52.54, -7.91) mm, rotated rx 180 ry 0 rz 90 deg; joints [71.755, -17.821, 85.781, 0, 22.04, 71.755]
  MoveL 6993 to (-34.54, -52.74, -8.31) mm, rotated rx 180 ry 0 rz 90 deg; joints [71.765, -17.773, 85.659, 0, 22.114, 71.765]
  MoveL 6994 to (-33.02, -52.6, -8.72) mm, rotated rx -180 ry 0 rz 90 deg; joints [71.785, -17.726, 85.543, 0, 22.183, 71.785]
  MoveL 6995 to (-31.58, -52.13, -9.13) mm, rotated rx 180 ry 0 rz 90 deg; joints [71.816, -17.683, 85.44, 0, 22.243, 71.816]
  MoveL 6996 to (-30.27, -51.36, -9.53) mm, rotated rx 180 ry 0 rz 90 deg; joints [71.855, -17.644, 85.353, 0, 22.29, 71.855]
  MoveL 6997 to (-29.17, -50.31, -9.94) mm, rotated rx -180 ry 0 rz 90 deg; joints [71.9, -17.61, 85.287, 0, 22.323, 71.9]
  MoveL 6998 to (-28.33, -49.05, -10.34) mm, rotated rx -180 ry 0 rz 90 deg; joints [71.95, -17.581, 85.243, 0, 22.338, 71.95]
  MoveL 6999 to (-27.81, -47.62, -10.75) mm, rotated rx 180 ry 0 rz 90 deg; joints [72.001, -17.559, 85.226, 0, 22.333, 72.001]
  MoveL 7000 to (-22.11, -25.59, -10.75) mm, rotated rx 180 ry 0 rz 90 deg; joints [72.772, -17.582, 85.316, 0, 22.266, 72.772]
  MoveC 7001 to (-22.01, -25.12, -10.75) mm, rotated rx -180 ry 0 rz 90 deg; joints [72.788, -17.583, 85.319, 0, 22.264, 72.788] to (-21.99, -24.64, -10.75) mm, rotated rx 180 ry 0 rz 90 deg; joints [72.804, -17.585, 85.328, 0, 22.257, 72.804]
  MoveC 7002 to (-22.91, -22.68, -10.75) mm, rotated rx 180 ry 0 rz 90 deg; joints [72.858, -17.612, 85.434, 0, 22.177, 72.858] to (-24.7, -21.45, -10.75) mm, rotated rx 180 ry 0 rz 90 deg; joints [72.88, -17.65, 85.585, 0, 22.065, 72.88]
  MoveC 7003 to (-25.15, -21.36, -10.75) mm, rotated rx 180 ry 0 rz 90 deg; joints [72.879, -17.658, 85.619, 0, 22.039, 72.879] to (-25.61, -21.39, -10.75) mm, rotated rx 180 ry 0 rz 90 deg; joints [72.873, -17.666, 85.65, 0, 22.016, 72.873]
  MoveL 7004 to (-30.8, -22.44, -10.75) mm, rotated rx 180 ry 0 rz 90 deg; joints [72.787, -17.75, 85.987, 0, 21.763, 72.787]
  MoveL 7005 to (-64.91, -29.5, -10.75) mm, rotated rx 180 ry 0 rz 90 deg; joints [72.201, -18.272, 88.166, 0, 20.107, 72.201]
  MoveL 7006 to (-70.48, -30.67, -10.75) mm, rotated rx -180 ry 0 rz 90 deg; joints [72.103, -18.353, 88.515, 0, 19.838, 72.103]
  MoveC 7007 to (-72.09, -31.6, -10.75) mm, rotated rx -180 ry 0 rz 90 deg; joints [72.055, -18.373, 88.602, 0, 19.771, 72.055] to (-72.81, -33.31, -10.75) mm, rotated rx 180 ry 0 rz 90 deg; joints [71.991, -18.376, 88.613, 0, 19.762, 71.991]
  MoveL 7008 to (-72.83, -33.64, -10.75) mm, rotated rx 180 ry 0 rz 90 deg; joints [71.979, -18.374, 88.608, 0, 19.767, 71.979]
  MoveL 7009 to (-72.84, -34.59, -10.75) mm, rotated rx 180 ry 0 rz 90 deg; joints [71.948, -18.37, 88.587, 0, 19.782, 71.948]
  MoveL 7010 to (-72.84, -68.7, -10.75) mm, rotated rx 180 ry 0 rz 90 deg; joints [70.824, -18.191, 87.817, 0, 20.374, 70.824]
  MoveL 7011 to (-72.82, -69.44, -10.75) mm, rotated rx 180 ry 0 rz 90 deg; joints [70.8, -18.187, 87.799, 0, 20.388, 70.8]
  MoveC 7012 to (-71.91, -71.53, -10.75) mm, rotated rx -180 ry 0 rz 90 deg; joints [70.742, -18.161, 87.688, 0, 20.473, 70.742] to (-69.79, -72.38, -10.75) mm, rotated rx -180 ry 0 rz 90 deg; joints [70.739, -18.122, 87.526, 0, 20.597, 70.739]
  MoveL 7013 to (-67.76, -72.36, -10.75) mm, rotated rx -180 ry 0 rz 90 deg; joints [70.762, -18.09, 87.389, 0, 20.701, 70.762]
  MoveL 7014 to (-38.38, -71.98, -10.75) mm, rotated rx -180 ry 0 rz 90 deg; joints [71.103, -17.602, 85.395, 0, 22.207, 71.103]
  MoveL 7015 to (-36.48, -71.94, -10.75) mm, rotated rx -180 ry 0 rz 90 deg; joints [71.125, -17.569, 85.265, 0, 22.304, 71.125]
  MoveC 7016 to (-34.61, -71.31, -10.75) mm, rotated rx 180 ry 0 rz 90 deg; joints [71.166, -17.54, 85.15, 0, 22.39, 71.166] to (-33.52, -69.65, -10.75) mm, rotated rx 180 ry 0 rz 90 deg; joints [71.231, -17.531, 85.114, 0, 22.417, 71.231]
  MoveL 7017 to (-27.81, -47.62, -10.75) mm, rotated rx 180 ry 0 rz 90 deg; joints [72.001, -17.559, 85.226, 0, 22.333, 72.001]
  MoveL 7018 to (-35.12, -45.73, -10.75) mm, rotated rx 180 ry 0 rz 90 deg; joints [71.985, -17.697, 85.775, 0, 21.922, 71.985]
  MoveL 7019 to (-35.12, -45.73, -7.75) mm, rotated rx 180 ry 0 rz 90 deg; joints [71.985, -17.852, 85.877, 0, 21.975, 71.985]
  Establecer velocidad (1000.0 mm/s)
  MoveL 7020 to (-35.12, -45.73, 10) mm, rotated rx 180 ry 0 rz 90 deg; joints [71.985, -18.764, 86.471, 0, 22.294, 71.985]
  Establecer velocidad (66.7 mm/s)
  MoveL 7021 to (-64.6, 35.83, 10) mm, rotated rx -180 ry 0 rz 90 deg; joints [74.392, -19.653, 90.161, 0, 19.492, 74.392]
  MoveL 7022 to (-64.6, 35.83, -7.5) mm, rotated rx 180 ry 0 rz 90 deg; joints [74.392, -18.738, 89.575, 0, 19.163, 74.392]
  MoveL 7023 to (-66.1, 36.02, -7.91) mm, rotated rx -180 ry 0 rz 90 deg; joints [74.384, -18.74, 89.666, 0, 19.074, 74.384]
  MoveL 7024 to (-67.61, 35.83, -8.31) mm, rotated rx 180 ry 0 rz 90 deg; joints [74.363, -18.74, 89.75, 0, 18.99, 74.363]
  MoveL 7025 to (-69.04, 35.32, -8.72) mm, rotated rx -180 ry 0 rz 90 deg; joints [74.332, -18.738, 89.823, 0, 18.916, 74.332]
  MoveL 7026 to (-70.32, 34.51, -9.13) mm, rotated rx 180 ry 0 rz 90 deg; joints [74.292, -18.732, 89.879, 0, 18.853, 74.292]
  MoveL 7027 to (-71.39, 33.43, -9.53) mm, rotated rx -180 ry 0 rz 90 deg; joints [74.246, -18.722, 89.917, 0, 18.806, 74.246]
  MoveL 7028 to (-72.2, 32.14, -9.94) mm, rotated rx 180 ry 0 rz 90 deg; joints [74.194, -18.708, 89.932, 0, 18.775, 74.194]
  MoveL 7029 to (-72.7, 30.7, -10.34) mm, rotated rx 180 ry 0 rz 90 deg; joints [74.141, -18.688, 89.925, 0, 18.763, 74.141]
  MoveL 7030 to (-72.84, 29.19, -10.75) mm, rotated rx -180 ry 0 rz 90 deg; joints [74.088, -18.662, 89.891, 0, 18.771, 74.088]
  MoveL 7031 to (-72.84, 3.32, -10.75) mm, rotated rx 180 ry 0 rz 90 deg; joints [73.214, -18.55, 89.384, 0, 19.166, 73.214]
  MoveL 7032 to (-72.82, 2.47, -10.75) mm, rotated rx -180 ry 0 rz 90 deg; joints [73.186, -18.546, 89.366, 0, 19.18, 73.186]
  MoveC 7033 to (-72.53, 1.27, -10.75) mm, rotated rx 180 ry 0 rz 90 deg; joints [73.148, -18.536, 89.322, 0, 19.214, 73.148] to (-71.76, 0.31, -10.75) mm, rotated rx 180 ry 0 rz 90 deg; joints [73.124, -18.52, 89.25, 0, 19.27, 73.124]
  MoveC 7034 to (-70.77, -0.28, -10.75) mm, rotated rx 180 ry 0 rz 90 deg; joints [73.114, -18.502, 89.172, 0, 19.33, 73.114] to (-69.64, -0.47, -10.75) mm, rotated rx -180 ry 0 rz 90 deg; joints [73.119, -18.485, 89.093, 0, 19.392, 73.119]
  MoveL 7035 to (-69.18, -0.39, -10.75) mm, rotated rx 180 ry 0 rz 90 deg; joints [73.127, -18.478, 89.064, 0, 19.414, 73.127]
  MoveL 7036 to (-68.7, -0.28, -10.75) mm, rotated rx -180 ry 0 rz 90 deg; joints [73.135, -18.471, 89.034, 0, 19.437, 73.135]
  MoveC 7037 to (-45.95, 5.05, -10.75) mm, rotated rx -180 ry 0 rz 90 deg; joints [73.54, -18.14, 87.601, 0, 20.539, 73.54] to (-23.22, 10.45, -10.75) mm, rotated rx 180 ry 0 rz 90 deg; joints [73.937, -17.788, 86.143, 0, 21.645, 73.937]
  MoveC 7038 to (-21.29, 12.14, -10.75) mm, rotated rx 180 ry 0 rz 90 deg; joints [74.01, -17.764, 86.043, 0, 21.721, 74.01] to (-21.15, 14.69, -10.75) mm, rotated rx 180 ry 0 rz 90 deg; joints [74.096, -17.774, 86.084, 0, 21.69, 74.096]
  MoveL 7039 to (-26.94, 31, -10.75) mm, rotated rx 180 ry 0 rz 90 deg; joints [74.58, -17.95, 86.804, 0, 21.146, 74.58]
  MoveC 7040 to (-27.45, 31.91, -10.75) mm, rotated rx -180 ry 0 rz 90 deg; joints [74.606, -17.962, 86.856, 0, 21.106, 74.606] to (-28.22, 32.62, -10.75) mm, rotated rx 180 ry 0 rz 90 deg; joints [74.622, -17.978, 86.923, 0, 21.056, 74.622]
  MoveC 7041 to (-48.37, 45.71, -10.75) mm, rotated rx -180 ry 0 rz 90 deg; joints [74.876, -18.361, 88.55, 0, 19.811, 74.876] to (-68.56, 58.72, -10.75) mm, rotated rx -180 ry 0 rz 90 deg; joints [75.134, -18.718, 90.149, 0, 18.569, 75.134]
  MoveC 7042 to (-70.78, 58.53, -10.75) mm, rotated rx 180 ry 0 rz 90 deg; joints [75.107, -18.75, 90.294, 0, 18.455, 75.107] to (-72.49, 57.11, -10.75) mm, rotated rx -180 ry 0 rz 90 deg; joints [75.043, -18.769, 90.384, 0, 18.385, 75.043]
  MoveC 7043 to (-72.76, 56.54, -10.75) mm, rotated rx 180 ry 0 rz 90 deg; joints [75.021, -18.771, 90.391, 0, 18.379, 75.021] to (-72.84, 55.91, -10.75) mm, rotated rx 180 ry 0 rz 90 deg; joints [74.999, -18.769, 90.385, 0, 18.384, 74.999]
  MoveL 7044 to (-72.84, 29.19, -10.75) mm, rotated rx -180 ry 0 rz 90 deg; joints [74.088, -18.662, 89.891, 0, 18.771, 74.088]
  MoveL 7045 to (-65.29, 29.19, -10.75) mm, rotated rx 180 ry 0 rz 90 deg; joints [74.161, -18.55, 89.385, 0, 19.165, 74.161]
  MoveL 7046 to (-65.29, 29.19, -7.75) mm, rotated rx -180 ry 0 rz 90 deg; joints [74.161, -18.707, 89.487, 0, 19.22, 74.161]
  Establecer velocidad (1000.0 mm/s)
  MoveL 7047 to (-65.29, 29.19, 10) mm, rotated rx -180 ry 0 rz 90 deg; joints [74.161, -19.635, 90.082, 0, 19.554, 74.161]
  Establecer velocidad (66.7 mm/s)
  MoveL 7048 to (-64.43, 35.83, 10) mm, rotated rx 180 ry 0 rz 90 deg; joints [74.393, -19.651, 90.15, 0, 19.501, 74.393]
  MoveL 7049 to (-64.43, 35.83, -7.75) mm, rotated rx 180 ry 0 rz 90 deg; joints [74.393, -18.722, 89.556, 0, 19.167, 74.393]
  MoveL 7050 to (-65.94, 36.02, -8.16) mm, rotated rx -180 ry 0 rz 90 deg; joints [74.385, -18.724, 89.647, 0, 19.078, 74.385]
  MoveL 7051 to (-67.45, 35.83, -8.56) mm, rotated rx -180 ry 0 rz 90 deg; joints [74.365, -18.725, 89.731, 0, 18.994, 74.365]
  MoveL 7052 to (-68.88, 35.32, -8.97) mm, rotated rx -180 ry 0 rz 90 deg; joints [74.334, -18.723, 89.803, 0, 18.919, 74.334]
  MoveL 7053 to (-70.16, 34.51, -9.38) mm, rotated rx -180 ry 0 rz 90 deg; joints [74.294, -18.717, 89.86, 0, 18.857, 74.294]
  MoveL 7054 to (-71.23, 33.43, -9.78) mm, rotated rx -180 ry 0 rz 90 deg; joints [74.247, -18.707, 89.897, 0, 18.81, 74.247]
  MoveL 7055 to (-72.03, 32.14, -10.19) mm, rotated rx 180 ry 0 rz 90 deg; joints [74.196, -18.692, 89.913, 0, 18.779, 74.196]
  MoveL 7056 to (-72.53, 30.7, -10.59) mm, rotated rx 180 ry 0 rz 90 deg; joints [74.142, -18.672, 89.905, 0, 18.767, 74.142]
  MoveL 7057 to (-72.67, 29.19, -11) mm, rotated rx 180 ry 0 rz 90 deg; joints [74.09, -18.647, 89.872, 0, 18.774, 74.09]
  MoveL 7058 to (-72.67, 3.32, -11) mm, rotated rx 180 ry 0 rz 90 deg; joints [73.216, -18.534, 89.364, 0, 19.17, 73.216]
  MoveL 7059 to (-72.65, 2.37, -11) mm, rotated rx 180 ry 0 rz 90 deg; joints [73.184, -18.53, 89.343, 0, 19.186, 73.184]
  MoveC 7060 to (-71.34, 0.27, -11) mm, rotated rx -180 ry 0 rz 90 deg; joints [73.127, -18.5, 89.213, 0, 19.287, 73.127] to (-68.91, -0.19, -11) mm, rotated rx -180 ry 0 rz 90 deg; joints [73.136, -18.462, 89.041, 0, 19.421, 73.136]
  MoveC 7061 to (-46.23, 5.13, -11) mm, rotated rx 180 ry 0 rz 90 deg; joints [73.54, -18.132, 87.614, 0, 20.519, 73.54] to (-23.58, 10.54, -11) mm, rotated rx 180 ry 0 rz 90 deg; joints [73.936, -17.782, 86.161, 0, 21.621, 73.936]
  MoveC 7062 to (-23.18, 10.66, -11) mm, rotated rx 180 ry 0 rz 90 deg; joints [73.944, -17.776, 86.136, 0, 21.64, 73.944] to (-22.79, 10.82, -11) mm, rotated rx 180 ry 0 rz 90 deg; joints [73.953, -17.77, 86.113, 0, 21.657, 73.953]
  MoveC 7063 to (-21.38, 12.5, -11) mm, rotated rx 180 ry 0 rz 90 deg; joints [74.022, -17.754, 86.048, 0, 21.706, 74.022] to (-21.31, 14.69, -11) mm, rotated rx 180 ry 0 rz 90 deg; joints [74.094, -17.764, 86.087, 0, 21.677, 74.094]
  MoveL 7064 to (-27.01, 30.72, -11) mm, rotated rx 180 ry 0 rz 90 deg; joints [74.57, -17.936, 86.794, 0, 21.142, 74.57]
  MoveC 7065 to (-27.39, 31.53, -11) mm, rotated rx 180 ry 0 rz 90 deg; joints [74.593, -17.946, 86.836, 0, 21.11, 74.593] to (-27.96, 32.22, -11) mm, rotated rx 180 ry 0 rz 90 deg; joints [74.611, -17.959, 86.889, 0, 21.071, 74.611]
  MoveL 7066 to (-28.63, 32.69, -11) mm, rotated rx 180 ry 0 rz 90 deg; joints [74.621, -17.972, 86.944, 0, 21.029, 74.621]
  MoveC 7067 to (-48.5, 45.62, -11) mm, rotated rx -180 ry 0 rz 90 deg; joints [74.872, -18.35, 88.549, 0, 19.801, 74.872] to (-68.43, 58.48, -11) mm, rotated rx -180 ry 0 rz 90 deg; joints [75.127, -18.702, 90.127, 0, 18.575, 75.127]
  MoveC 7068 to (-70.36, 58.4, -11) mm, rotated rx 180 ry 0 rz 90 deg; joints [75.106, -18.73, 90.255, 0, 18.475, 75.106] to (-71.97, 57.33, -11) mm, rotated rx 180 ry 0 rz 90 deg; joints [75.055, -18.749, 90.344, 0, 18.405, 75.055]
  MoveL 7069 to (-72.17, 57.1, -11) mm, rotated rx 180 ry 0 rz 90 deg; joints [75.046, -18.751, 90.353, 0, 18.398, 75.046]
  MoveC 7070 to (-72.54, 56.48, -11) mm, rotated rx -180 ry 0 rz 90 deg; joints [75.021, -18.754, 90.367, 0, 18.387, 75.021] to (-72.67, 55.77, -11) mm, rotated rx 180 ry 0 rz 90 deg; joints [74.995, -18.753, 90.363, 0, 18.39, 74.995]
  MoveL 7071 to (-72.67, 29.19, -11) mm, rotated rx 180 ry 0 rz 90 deg; joints [74.09, -18.647, 89.872, 0, 18.774, 74.09]
  MoveL 7072 to (-65.12, 29.19, -11) mm, rotated rx 180 ry 0 rz 90 deg; joints [74.162, -18.535, 89.366, 0, 19.169, 74.162]
  MoveL 7073 to (-65.12, 29.19, -8) mm, rotated rx 180 ry 0 rz 90 deg; joints [74.162, -18.691, 89.468, 0, 19.224, 74.162]
  Establecer velocidad (1000.0 mm/s)
  MoveL 7074 to (-65.12, 29.19, 10) mm, rotated rx -180 ry 0 rz 90 deg; joints [74.162, -19.633, 90.07, 0, 19.562, 74.162]
  Establecer velocidad (66.7 mm/s)
  MoveL 7075 to (-39.92, -32.91, 10) mm, rotated rx 180 ry 0 rz 90 deg; joints [72.352, -18.919, 87.085, 0, 21.834, 72.352]
  MoveL 7076 to (-39.92, -32.91, -7.75) mm, rotated rx 180 ry 0 rz 90 deg; joints [72.352, -18.004, 86.492, 0, 21.512, 72.352]
  MoveL 7077 to (-40.04, -31.4, -8.16) mm, rotated rx -180 ry 0 rz 90 deg; joints [72.4, -17.993, 86.519, 0, 21.474, 72.4]
  MoveL 7078 to (-40.53, -29.96, -8.56) mm, rotated rx -180 ry 0 rz 90 deg; joints [72.442, -17.988, 86.57, 0, 21.417, 72.442]
  MoveL 7079 to (-41.32, -28.66, -8.97) mm, rotated rx 180 ry 0 rz 90 deg; joints [72.476, -17.987, 86.639, 0, 21.348, 72.476]
  MoveL 7080 to (-42.37, -27.57, -9.38) mm, rotated rx 180 ry 0 rz 90 deg; joints [72.501, -17.989, 86.721, 0, 21.268, 72.501]
  MoveL 7081 to (-43.65, -26.74, -9.78) mm, rotated rx -180 ry 0 rz 90 deg; joints [72.515, -17.994, 86.813, 0, 21.181, 72.515]
  MoveL 7082 to (-45.07, -26.21, -10.19) mm, rotated rx -180 ry 0 rz 90 deg; joints [72.518, -17.999, 86.908, 0, 21.091, 72.518]
  MoveL 7083 to (-46.58, -26.01, -10.59) mm, rotated rx -180 ry 0 rz 90 deg; joints [72.509, -18.004, 87.001, 0, 21.003, 72.509]
  MoveL 7084 to (-48.08, -26.18, -11) mm, rotated rx -180 ry 0 rz 90 deg; joints [72.487, -18.007, 87.087, 0, 20.92, 72.487]
  MoveL 7085 to (-63.97, -29.45, -11) mm, rotated rx -180 ry 0 rz 90 deg; joints [72.213, -18.245, 88.094, 0, 20.151, 72.213]
  MoveL 7086 to (-70.33, -30.79, -11) mm, rotated rx -180 ry 0 rz 90 deg; joints [72.101, -18.337, 88.494, 0, 19.844, 72.101]
  MoveC 7087 to (-71.9, -31.69, -11) mm, rotated rx 180 ry 0 rz 90 deg; joints [72.054, -18.357, 88.579, 0, 19.777, 72.054] to (-72.64, -33.34, -11) mm, rotated rx 180 ry 0 rz 90 deg; joints [71.992, -18.36, 88.593, 0, 19.767, 71.992]
  MoveC 7088 to (-72.67, -33.63, -11) mm, rotated rx 180 ry 0 rz 90 deg; joints [71.982, -18.359, 88.588, 0, 19.771, 71.982] to (-72.67, -33.93, -11) mm, rotated rx -180 ry 0 rz 90 deg; joints [71.972, -18.357, 88.582, 0, 19.775, 71.972]
  MoveL 7089 to (-72.67, -69.23, -11) mm, rotated rx 180 ry 0 rz 90 deg; joints [70.809, -18.173, 87.785, 0, 20.388, 70.809]
  MoveC 7090 to (-72.34, -70.6, -11) mm, rotated rx 180 ry 0 rz 90 deg; joints [70.768, -18.16, 87.731, 0, 20.429, 70.768] to (-71.42, -71.67, -11) mm, rotated rx -180 ry 0 rz 90 deg; joints [70.743, -18.139, 87.644, 0, 20.495, 70.743]
  MoveC 7091 to (-70.58, -72.09, -11) mm, rotated rx -180 ry 0 rz 90 deg; joints [70.739, -18.124, 87.577, 0, 20.546, 70.739] to (-69.65, -72.22, -11) mm, rotated rx 180 ry 0 rz 90 deg; joints [70.745, -18.108, 87.512, 0, 20.596, 70.745]
  MoveC 7092 to (-53.07, -72.03, -11) mm, rotated rx 180 ry 0 rz 90 deg; joints [70.939, -17.839, 86.393, 0, 21.446, 70.939] to (-36.48, -71.78, -11) mm, rotated rx -180 ry 0 rz 90 deg; joints [71.131, -17.557, 85.26, 0, 22.297, 71.131]
  MoveC 7093 to (-34.69, -71.13, -11) mm, rotated rx -180 ry 0 rz 90 deg; joints [71.171, -17.53, 85.152, 0, 22.378, 71.171] to (-33.64, -69.55, -11) mm, rotated rx 180 ry 0 rz 90 deg; joints [71.233, -17.521, 85.116, 0, 22.405, 71.233]
  MoveL 7094 to (-31.7, -62.07, -11) mm, rotated rx 180 ry 0 rz 90 deg; joints [71.494, -17.531, 85.156, 0, 22.375, 71.494]
  MoveL 7095 to (-22.24, -25.45, -11) mm, rotated rx -180 ry 0 rz 90 deg; joints [72.775, -17.572, 85.319, 0, 22.253, 72.775]
  MoveC 7096 to (-22.18, -25.05, -11) mm, rotated rx 180 ry 0 rz 90 deg; joints [72.789, -17.573, 85.324, 0, 22.249, 72.789] to (-22.23, -24.64, -11) mm, rotated rx 180 ry 0 rz 90 deg; joints [72.802, -17.576, 85.336, 0, 22.24, 72.802]
  MoveC 7097 to (-23.13, -22.87, -11) mm, rotated rx -180 ry 0 rz 90 deg; joints [72.85, -17.602, 85.437, 0, 22.165, 72.85] to (-24.75, -21.71, -11) mm, rotated rx 180 ry 0 rz 90 deg; joints [72.871, -17.636, 85.575, 0, 22.062, 72.871]
  MoveC 7098 to (-25.28, -21.59, -11) mm, rotated rx 180 ry 0 rz 90 deg; joints [72.87, -17.646, 85.614, 0, 22.032, 72.87] to (-25.83, -21.62, -11) mm, rotated rx 180 ry 0 rz 90 deg; joints [72.864, -17.656, 85.652, 0, 22.004, 72.864]
  MoveL 7099 to (-30.8, -22.62, -11) mm, rotated rx 180 ry 0 rz 90 deg; joints [72.781, -17.736, 85.975, 0, 21.761, 72.781]
  MoveL 7100 to (-48.08, -26.18, -11) mm, rotated rx -180 ry 0 rz 90 deg; joints [72.487, -18.007, 87.087, 0, 20.92, 72.487]
  MoveL 7101 to (-46.56, -33.58, -11) mm, rotated rx 180 ry 0 rz 90 deg; joints [72.261, -17.943, 86.822, 0, 21.121, 72.261]
  MoveL 7102 to (-46.56, -33.58, -8) mm, rotated rx -180 ry 0 rz 90 deg; joints [72.261, -18.098, 86.924, 0, 21.174, 72.261]
  Establecer velocidad (1000.0 mm/s)
  MoveL 7103 to (-46.56, -33.58, 10) mm, rotated rx 180 ry 0 rz 90 deg; joints [72.261, -19.028, 87.526, 0, 21.502, 72.261]
  Establecer velocidad (66.7 mm/s)
  MoveL 7104 to (14.72, -62.67, 10) mm, rotated rx 180 ry 0 rz 90 deg; joints [71.962, -17.727, 82.567, 0, 25.159, 71.962]
  MoveL 7105 to (14.72, -62.67, -7.75) mm, rotated rx -180 ry 0 rz 90 deg; joints [71.962, -16.828, 81.971, 0, 24.856, 71.962]
  MoveL 7106 to (14.59, -64.18, -8.16) mm, rotated rx 180 ry 0 rz 90 deg; joints [71.914, -16.8, 81.931, 0, 24.869, 71.914]
  MoveL 7107 to (14.84, -65.68, -8.56) mm, rotated rx -180 ry 0 rz 90 deg; joints [71.869, -16.765, 81.865, 0, 24.9, 71.869]
  MoveL 7108 to (15.4, -67.09, -8.97) mm, rotated rx 180 ry 0 rz 90 deg; joints [71.831, -16.724, 81.777, 0, 24.947, 71.831]
  MoveL 7109 to (16.27, -68.34, -9.38) mm, rotated rx -180 ry 0 rz 90 deg; joints [71.8, -16.678, 81.671, 0, 25.007, 71.8]
  MoveL 7110 to (17.38, -69.37, -9.78) mm, rotated rx 180 ry 0 rz 90 deg; joints [71.78, -16.628, 81.552, 0, 25.077, 71.78]
  MoveL 7111 to (18.7, -70.12, -10.19) mm, rotated rx -180 ry 0 rz 90 deg; joints [71.77, -16.576, 81.424, 0, 25.152, 71.77]
  MoveL 7112 to (20.16, -70.57, -10.59) mm, rotated rx -180 ry 0 rz 90 deg; joints [71.771, -16.524, 81.294, 0, 25.229, 71.771]
  MoveL 7113 to (21.67, -70.65, -11) mm, rotated rx 180 ry 0 rz 90 deg; joints [71.784, -16.472, 81.169, 0, 25.304, 71.784]
  MoveC 7114 to (31.32, -70.25, -11) mm, rotated rx 180 ry 0 rz 90 deg; joints [71.895, -16.278, 80.475, 0, 25.803, 71.895] to (40.96, -69.77, -11) mm, rotated rx 180 ry 0 rz 90 deg; joints [72.007, -16.081, 79.777, 0, 26.303, 72.007]
  MoveC 7115 to (43.13, -66.89, -11) mm, rotated rx -180 ry 0 rz 90 deg; joints [72.118, -16.055, 79.686, 0, 26.369, 72.118] to (43.26, -63.28, -11) mm, rotated rx -180 ry 0 rz 90 deg; joints [72.231, -16.076, 79.762, 0, 26.314, 72.231]
  MoveC 7116 to (33.47, -51.21, -11) mm, rotated rx -180 ry 0 rz 90 deg; joints [72.509, -16.36, 80.765, 0, 25.595, 72.509] to (23.55, -39.26, -11) mm, rotated rx -180 ry 0 rz 90 deg; joints [72.787, -16.635, 81.76, 0, 24.875, 72.787]
  MoveC 7117 to (23.14, -38.82, -11) mm, rotated rx -180 ry 0 rz 90 deg; joints [72.797, -16.646, 81.8, 0, 24.846, 72.797] to (22.68, -38.41, -11) mm, rotated rx 180 ry 0 rz 90 deg; joints [72.806, -16.658, 81.842, 0, 24.816, 72.806]
  MoveL 7118 to (13.64, -30.97, -11) mm, rotated rx -180 ry 0 rz 90 deg; joints [72.953, -16.88, 82.66, 0, 24.22, 72.953]
  MoveC 7119 to (10.88, -30.5, -11) mm, rotated rx 180 ry 0 rz 90 deg; joints [72.941, -16.935, 82.868, 0, 24.067, 72.941] to (8.57, -32.08, -11) mm, rotated rx -180 ry 0 rz 90 deg; joints [72.868, -16.97, 82.999, 0, 23.972, 72.868]
  MoveL 7120 to (8.39, -32.69, -11) mm, rotated rx 180 ry 0 rz 90 deg; joints [72.847, -16.97, 82.998, 0, 23.972, 72.847]
  MoveL 7121 to (-0.86, -66.81, -11) mm, rotated rx 180 ry 0 rz 90 deg; joints [71.671, -16.938, 82.88, 0, 24.059, 71.671]
  MoveL 7122 to (-1.09, -67.76, -11) mm, rotated rx -180 ry 0 rz 90 deg; joints [71.638, -16.937, 82.873, 0, 24.063, 71.638]
  MoveC 7123 to (-0.12, -70.25, -11) mm, rotated rx 180 ry 0 rz 90 deg; joints [71.57, -16.902, 82.745, 0, 24.157, 71.57] to (2.37, -71.24, -11) mm, rotated rx -180 ry 0 rz 90 deg; joints [71.565, -16.848, 82.544, 0, 24.304, 71.565]
  MoveC 7124 to (12.02, -70.98, -11) mm, rotated rx 180 ry 0 rz 90 deg; joints [71.674, -16.662, 81.858, 0, 24.804, 71.674] to (21.67, -70.65, -11) mm, rotated rx 180 ry 0 rz 90 deg; joints [71.784, -16.472, 81.169, 0, 25.304, 71.784]
  MoveL 7125 to (21.38, -63.1, -11) mm, rotated rx 180 ry 0 rz 90 deg; joints [72.017, -16.528, 81.368, 0, 25.159, 72.017]
  MoveL 7126 to (21.38, -63.1, -8) mm, rotated rx 180 ry 0 rz 90 deg; joints [72.017, -16.68, 81.471, 0, 25.208, 72.017]
  Establecer velocidad (1000.0 mm/s)
  MoveL 7127 to (21.38, -63.1, 10) mm, rotated rx 180 ry 0 rz 90 deg; joints [72.017, -17.59, 82.076, 0, 25.513, 72.017]
  Establecer velocidad (66.7 mm/s)
  MoveL 7128 to (35.13, 17.64, 10) mm, rotated rx -180 ry 0 rz 90 deg; joints [74.7, -17.8, 82.831, 0, 24.969, 74.7]
  MoveL 7129 to (35.13, 17.64, -7.75) mm, rotated rx 180 ry 0 rz 90 deg; joints [74.7, -16.9, 82.235, 0, 24.664, 74.7]
  MoveL 7130 to (35.32, 19.14, -8.16) mm, rotated rx 180 ry 0 rz 90 deg; joints [74.75, -16.884, 82.238, 0, 24.646, 74.75]
  MoveL 7131 to (35.14, 20.65, -8.56) mm, rotated rx 180 ry 0 rz 90 deg; joints [74.796, -16.875, 82.267, 0, 24.608, 74.796]
  MoveL 7132 to (34.64, 22.09, -8.97) mm, rotated rx 180 ry 0 rz 90 deg; joints [74.838, -16.872, 82.318, 0, 24.554, 74.838]
  MoveL 7133 to (33.83, 23.37, -9.38) mm, rotated rx -180 ry 0 rz 90 deg; joints [74.872, -16.874, 82.389, 0, 24.485, 74.872]
  MoveL 7134 to (32.75, 24.44, -9.78) mm, rotated rx -180 ry 0 rz 90 deg; joints [74.897, -16.88, 82.474, 0, 24.406, 74.897]
  MoveL 7135 to (31.47, 25.26, -10.19) mm, rotated rx 180 ry 0 rz 90 deg; joints [74.912, -16.889, 82.57, 0, 24.32, 74.912]
  MoveL 7136 to (30.03, 25.76, -10.59) mm, rotated rx 180 ry 0 rz 90 deg; joints [74.916, -16.899, 82.67, 0, 24.229, 74.916]
  MoveL 7137 to (28.52, 25.9, -11) mm, rotated rx -180 ry 0 rz 90 deg; joints [74.907, -16.909, 82.768, 0, 24.141, 74.907]
  MoveC 7138 to (21.4, 25.9, -11) mm, rotated rx -180 ry 0 rz 90 deg; joints [74.845, -17.046, 83.283, 0, 23.763, 74.845] to (14.27, 25.85, -11) mm, rotated rx -180 ry 0 rz 90 deg; joints [74.781, -17.18, 83.794, 0, 23.386, 74.781]
  MoveC 7139 to (12.09, 25.07, -11) mm, rotated rx 180 ry 0 rz 90 deg; joints [74.736, -17.217, 83.935, 0, 23.282, 74.736] to (10.86, 23.1, -11) mm, rotated rx -180 ry 0 rz 90 deg; joints [74.662, -17.23, 83.984, 0, 23.246, 74.662]
  MoveC 7140 to (10.81, 22.39, -11) mm, rotated rx -180 ry 0 rz 90 deg; joints [74.638, -17.227, 83.974, 0, 23.254, 74.638] to (10.96, 21.7, -11) mm, rotated rx -180 ry 0 rz 90 deg; joints [74.617, -17.221, 83.95, 0, 23.271, 74.617]
  MoveL 7141 to (14.59, 11.85, -11) mm, rotated rx -180 ry 0 rz 90 deg; joints [74.332, -17.102, 83.494, 0, 23.608, 74.332]
  MoveL 7142 to (14.81, 11.27, -11) mm, rotated rx 180 ry 0 rz 90 deg; joints [74.315, -17.094, 83.466, 0, 23.628, 74.315]
  MoveC 7143 to (15.22, 10.54, -11) mm, rotated rx 180 ry 0 rz 90 deg; joints [74.295, -17.083, 83.422, 0, 23.661, 74.295] to (15.82, 9.95, -11) mm, rotated rx 180 ry 0 rz 90 deg; joints [74.282, -17.068, 83.367, 0, 23.701, 74.282]
  MoveL 7144 to (28.18, 0.75, -11) mm, rotated rx -180 ry 0 rz 90 deg; joints [74.099, -16.779, 82.287, 0, 24.492, 74.099]
  MoveC 7145 to (29.34, 0.21, -11) mm, rotated rx 180 ry 0 rz 90 deg; joints [74.093, -16.753, 82.192, 0, 24.561, 74.093] to (30.62, 0.18, -11) mm, rotated rx -180 ry 0 rz 90 deg; joints [74.103, -16.728, 82.098, 0, 24.63, 74.103]
  MoveC 7146 to (32.09, 0.76, -11) mm, rotated rx 180 ry 0 rz 90 deg; joints [74.135, -16.702, 82.003, 0, 24.699, 74.135] to (33.23, 1.86, -11) mm, rotated rx 180 ry 0 rz 90 deg; joints [74.18, -16.685, 81.942, 0, 24.743, 74.18]
  MoveL 7147 to (35.54, 5.21, -11) mm, rotated rx 180 ry 0 rz 90 deg; joints [74.308, -16.658, 81.843, 0, 24.815, 74.308]
  MoveL 7148 to (43.96, 17.53, -11) mm, rotated rx 180 ry 0 rz 90 deg; joints [74.773, -16.557, 81.476, 0, 25.081, 74.773]
  MoveL 7149 to (45.01, 19.1, -11) mm, rotated rx 180 ry 0 rz 90 deg; joints [74.832, -16.545, 81.43, 0, 25.115, 74.832]
  MoveL 7150 to (45.39, 19.95, -11) mm, rotated rx 180 ry 0 rz 90 deg; joints [74.862, -16.542, 81.419, 0, 25.123, 74.862]
  MoveL 7151 to (45.39, 21.47, -11) mm, rotated rx -180 ry 0 rz 90 deg; joints [74.911, -16.55, 81.449, 0, 25.101, 74.911]
  MoveC 7152 to (44.58, 23.91, -11) mm, rotated rx -180 ry 0 rz 90 deg; joints [74.981, -16.58, 81.557, 0, 25.022, 74.981] to (42.77, 25.75, -11) mm, rotated rx -180 ry 0 rz 90 deg; joints [75.025, -16.626, 81.726, 0, 24.9, 75.025]
  MoveC 7153 to (35.65, 25.85, -11) mm, rotated rx 180 ry 0 rz 90 deg; joints [74.967, -16.769, 82.249, 0, 24.52, 74.967] to (28.52, 25.9, -11) mm, rotated rx -180 ry 0 rz 90 deg; joints [74.907, -16.909, 82.768, 0, 24.141, 74.907]
  MoveL 7154 to (28.49, 18.35, -11) mm, rotated rx 180 ry 0 rz 90 deg; joints [74.665, -16.869, 82.621, 0, 24.248, 74.665]
  MoveL 7155 to (28.49, 18.35, -8) mm, rotated rx 180 ry 0 rz 90 deg; joints [74.665, -17.022, 82.724, 0, 24.298, 74.665]
  Establecer velocidad (1000.0 mm/s)
  MoveL 7156 to (28.49, 18.35, 10) mm, rotated rx 180 ry 0 rz 90 deg; joints [74.665, -17.936, 83.328, 0, 24.609, 74.665]
  Establecer velocidad (66.7 mm/s)
  MoveL 7157 to (-0.04, 59.13, 10) mm, rotated rx 180 ry 0 rz 90 deg; joints [75.744, -18.68, 86.139, 0, 22.541, 75.744]
  MoveL 7158 to (-0.04, 59.13, -7.75) mm, rotated rx 180 ry 0 rz 90 deg; joints [75.744, -17.768, 85.545, 0, 22.223, 75.744]
  MoveL 7159 to (1.24, 58.3, -8.16) mm, rotated rx 180 ry 0 rz 90 deg; joints [75.728, -17.721, 85.426, 0, 22.295, 75.728]
  MoveL 7160 to (2.68, 57.81, -8.56) mm, rotated rx 180 ry 0 rz 90 deg; joints [75.724, -17.672, 85.302, 0, 22.37, 75.724]
  MoveL 7161 to (4.19, 57.67, -8.97) mm, rotated rx 180 ry 0 rz 90 deg; joints [75.732, -17.623, 85.178, 0, 22.445, 75.732]
  MoveL 7162 to (5.69, 57.86, -9.38) mm, rotated rx 180 ry 0 rz 90 deg; joints [75.751, -17.576, 85.061, 0, 22.515, 75.751]
  MoveL 7163 to (7.12, 58.39, -9.78) mm, rotated rx -180 ry 0 rz 90 deg; joints [75.78, -17.532, 84.956, 0, 22.577, 75.78]
  MoveL 7164 to (8.38, 59.24, -10.19) mm, rotated rx 180 ry 0 rz 90 deg; joints [75.818, -17.492, 84.867, 0, 22.625, 75.818]
  MoveL 7165 to (9.43, 60.34, -10.59) mm, rotated rx -180 ry 0 rz 90 deg; joints [75.863, -17.457, 84.799, 0, 22.659, 75.863]
  MoveL 7166 to (10.17, 61.67, -11) mm, rotated rx -180 ry 0 rz 90 deg; joints [75.912, -17.429, 84.756, 0, 22.673, 75.912]
  MoveL 7167 to (14.12, 70.67, -11) mm, rotated rx 180 ry 0 rz 90 deg; joints [76.24, -17.398, 84.633, 0, 22.765, 76.24]
  MoveC 7168 to (-1.53, 71.15, -11) mm, rotated rx -180 ry 0 rz 90 deg; joints [76.129, -17.681, 85.752, 0, 21.928, 76.129] to (-17.18, 71.54, -11) mm, rotated rx -180 ry 0 rz 90 deg; joints [76.013, -17.951, 86.856, 0, 21.095, 76.013]
  MoveC 7169 to (-19.42, 68.79, -11) mm, rotated rx -180 ry 0 rz 90 deg; joints [75.902, -17.977, 86.964, 0, 21.013, 75.902] to (-19.13, 65.26, -11) mm, rotated rx -180 ry 0 rz 90 deg; joints [75.787, -17.958, 86.882, 0, 21.076, 75.787]
  MoveL 7170 to (-8.05, 58.09, -11) mm, rotated rx -180 ry 0 rz 90 deg; joints [75.643, -17.737, 85.98, 0, 21.757, 75.643]
  MoveL 7171 to (-6.93, 57.33, -11) mm, rotated rx -180 ry 0 rz 90 deg; joints [75.627, -17.714, 85.888, 0, 21.826, 75.627]
